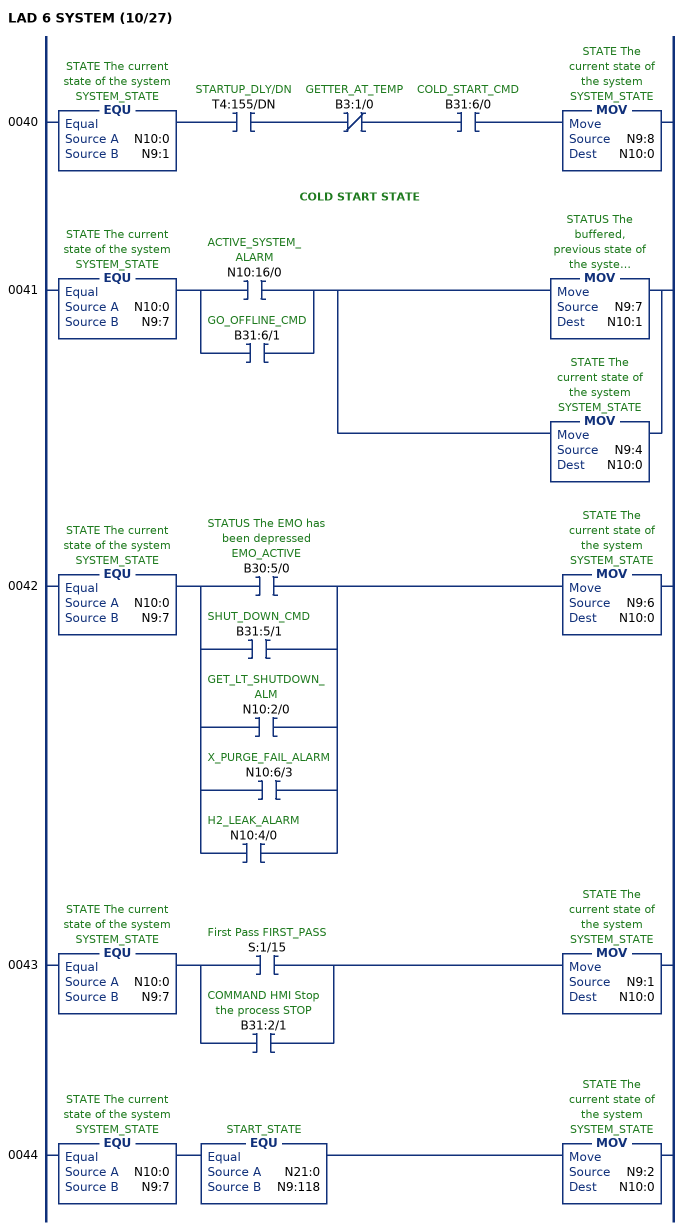
% Rung: 40 %
SOR EQU N10:0 N9:1 XIC T4:155/DN XIO B3:1/0 XIC B31:6/0 MOV N9:8 N10:0 EOR
%   N10:0  SYSTEM_STATE  "STATE The current state of the system" %
%   N9:1  SYSTEM_STANDBY  "STATE System Process" %
%   T4:155  STARTUP_DLY %
%   B3:1/0  GETTER_AT_TEMP %
%   B31:6/0  COLD_START_CMD %
%   N9:8  SYSTEM_SUPPLEMENTAL %
% Rung: 41 %
% TITLE: COLD START STATE %
SOR EQU N10:0 N9:7 BST XIC N10:16/0 NXB XIC B31:6/1 BND BST MOV N9:7 N10:1 NXB MOV N9:4 N10:0 BND EOR
%   N10:0  SYSTEM_STATE  "STATE The current state of the system" %
%   N9:7  SYSTEM_COLD_START %
%   N10:16/0  ACTIVE_SYSTEM_ALARM %
%   B31:6/1  GO_OFFLINE_CMD %
%   N10:1  SYSTEM_STATE_BUFFER  "STATUS The buffered, previous state of the system" %
%   N9:4  SYSTEM_ALARM  "STATE System Alarm" %
% Rung: 42 %
SOR EQU N10:0 N9:7 BST XIC B30:5/0 NXB XIC B31:5/1 NXB XIC N10:2/0 NXB XIC N10:6/3 NXB XIC N10:4/0 BND MOV N9:6 N10:0 EOR
%   N10:0  SYSTEM_STATE  "STATE The current state of the system" %
%   N9:7  SYSTEM_COLD_START %
%   B30:5/0  EMO_ACTIVE  "STATUS The EMO has been depressed" %
%   B31:5/1  SHUT_DOWN_CMD %
%   N10:2/0  GET_LT_SHUTDOWN_ALM %
%   N10:6/3  X_PURGE_FAIL_ALARM %
%   N10:4/0  H2_LEAK_ALARM %
%   N9:6  SYSTEM_PURGE %
% Rung: 43 %
SOR EQU N10:0 N9:7 BST XIC S:1/15 NXB XIC B31:2/1 BND MOV N9:1 N10:0 EOR
%   N10:0  SYSTEM_STATE  "STATE The current state of the system" %
%   N9:7  SYSTEM_COLD_START %
%   S:1/15  FIRST_PASS  "First Pass" %
%   B31:2/1  STOP  "COMMAND HMI Stop the process" %
%   N9:1  SYSTEM_STANDBY  "STATE System Process" %
% Rung: 44 %
SOR EQU N10:0 N9:7 EQU N21:0 N9:118 MOV N9:2 N10:0 EOR
%   N10:0  SYSTEM_STATE  "STATE The current state of the system" %
%   N9:7  SYSTEM_COLD_START %
%   N21:0  START_STATE %
%   N9:118  START_DONE %
%   N9:2  SYSTEM_PROCESS  "STATE System Process" %

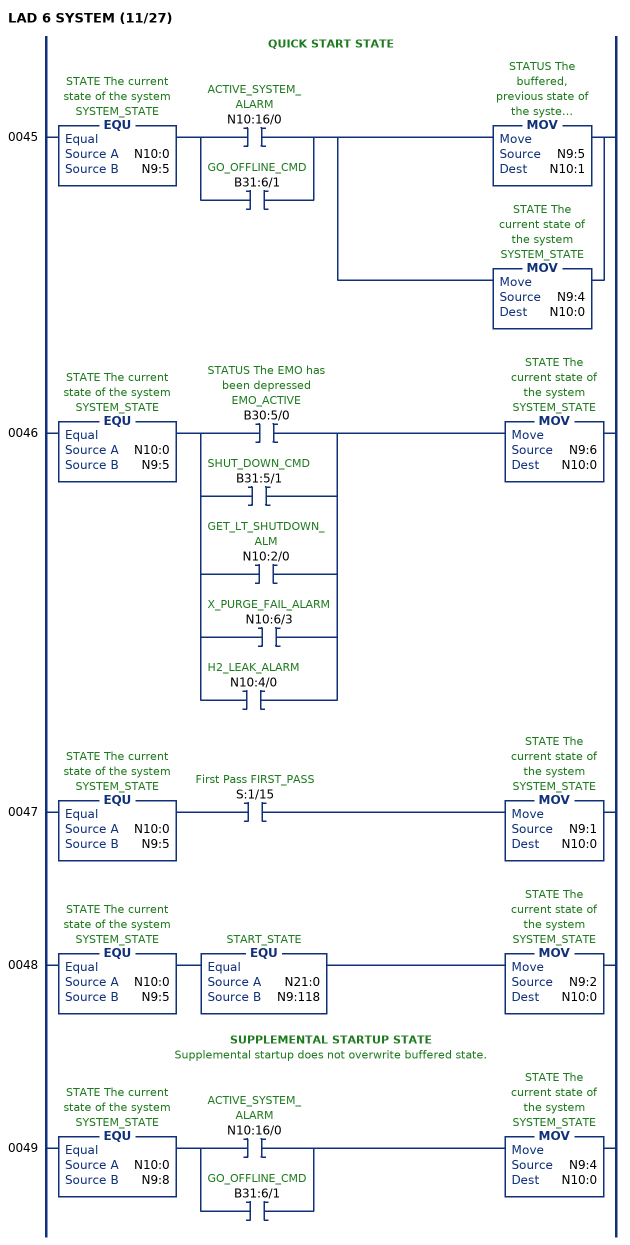
% Rung: 45 %
% TITLE: QUICK START STATE %
SOR EQU N10:0 N9:5 BST XIC N10:16/0 NXB XIC B31:6/1 BND BST MOV N9:5 N10:1 NXB MOV N9:4 N10:0 BND EOR
%   N10:0  SYSTEM_STATE  "STATE The current state of the system" %
%   N9:5  SYSTEM_QUICK_START %
%   N10:16/0  ACTIVE_SYSTEM_ALARM %
%   B31:6/1  GO_OFFLINE_CMD %
%   N10:1  SYSTEM_STATE_BUFFER  "STATUS The buffered, previous state of the system" %
%   N9:4  SYSTEM_ALARM  "STATE System Alarm" %
% Rung: 46 %
SOR EQU N10:0 N9:5 BST XIC B30:5/0 NXB XIC B31:5/1 NXB XIC N10:2/0 NXB XIC N10:6/3 NXB XIC N10:4/0 BND MOV N9:6 N10:0 EOR
%   N10:0  SYSTEM_STATE  "STATE The current state of the system" %
%   N9:5  SYSTEM_QUICK_START %
%   B30:5/0  EMO_ACTIVE  "STATUS The EMO has been depressed" %
%   B31:5/1  SHUT_DOWN_CMD %
%   N10:2/0  GET_LT_SHUTDOWN_ALM %
%   N10:6/3  X_PURGE_FAIL_ALARM %
%   N10:4/0  H2_LEAK_ALARM %
%   N9:6  SYSTEM_PURGE %
% Rung: 47 %
SOR EQU N10:0 N9:5 XIC S:1/15 MOV N9:1 N10:0 EOR
%   N10:0  SYSTEM_STATE  "STATE The current state of the system" %
%   N9:5  SYSTEM_QUICK_START %
%   S:1/15  FIRST_PASS  "First Pass" %
%   N9:1  SYSTEM_STANDBY  "STATE System Process" %
% Rung: 48 %
SOR EQU N10:0 N9:5 EQU N21:0 N9:118 MOV N9:2 N10:0 EOR
%   N10:0  SYSTEM_STATE  "STATE The current state of the system" %
%   N9:5  SYSTEM_QUICK_START %
%   N21:0  START_STATE %
%   N9:118  START_DONE %
%   N9:2  SYSTEM_PROCESS  "STATE System Process" %
% Rung: 49 %
% TITLE: SUPPLEMENTAL STARTUP STATE %
% Supplemental startup does not overwrite buffered state. %
SOR EQU N10:0 N9:8 BST XIC N10:16/0 NXB XIC B31:6/1 BND MOV N9:4 N10:0 EOR
%   N10:0  SYSTEM_STATE  "STATE The current state of the system" %
%   N9:8  SYSTEM_SUPPLEMENTAL %
%   N10:16/0  ACTIVE_SYSTEM_ALARM %
%   B31:6/1  GO_OFFLINE_CMD %
%   N9:4  SYSTEM_ALARM  "STATE System Alarm" %

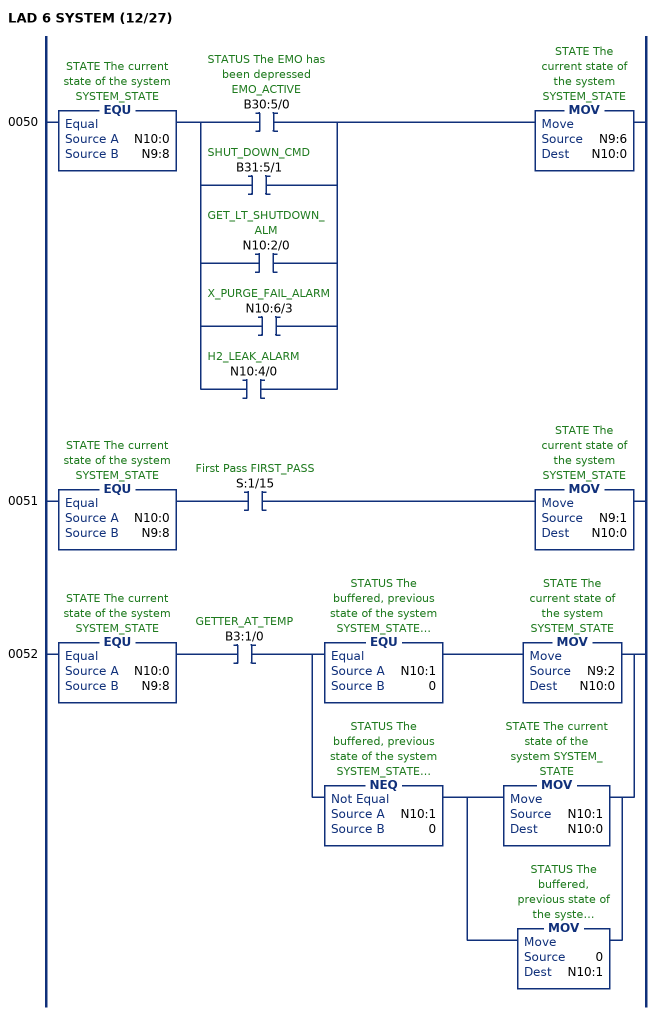
% Rung: 50 %
SOR EQU N10:0 N9:8 BST XIC B30:5/0 NXB XIC B31:5/1 NXB XIC N10:2/0 NXB XIC N10:6/3 NXB XIC N10:4/0 BND MOV N9:6 N10:0 EOR
%   N10:0  SYSTEM_STATE  "STATE The current state of the system" %
%   N9:8  SYSTEM_SUPPLEMENTAL %
%   B30:5/0  EMO_ACTIVE  "STATUS The EMO has been depressed" %
%   B31:5/1  SHUT_DOWN_CMD %
%   N10:2/0  GET_LT_SHUTDOWN_ALM %
%   N10:6/3  X_PURGE_FAIL_ALARM %
%   N10:4/0  H2_LEAK_ALARM %
%   N9:6  SYSTEM_PURGE %
% Rung: 51 %
SOR EQU N10:0 N9:8 XIC S:1/15 MOV N9:1 N10:0 EOR
%   N10:0  SYSTEM_STATE  "STATE The current state of the system" %
%   N9:8  SYSTEM_SUPPLEMENTAL %
%   S:1/15  FIRST_PASS  "First Pass" %
%   N9:1  SYSTEM_STANDBY  "STATE System Process" %
% Rung: 52 %
SOR EQU N10:0 N9:8 XIC B3:1/0 BST EQU N10:1 0 MOV N9:2 N10:0 NXB NEQ N10:1 0 BST MOV N10:1 N10:0 NXB MOV 0 N10:1 BND BND EOR
%   N10:0  SYSTEM_STATE  "STATE The current state of the system" %
%   N9:8  SYSTEM_SUPPLEMENTAL %
%   B3:1/0  GETTER_AT_TEMP %
%   N10:1  SYSTEM_STATE_BUFFER  "STATUS The buffered, previous state of the system" %
%   N9:2  SYSTEM_PROCESS  "STATE System Process" %

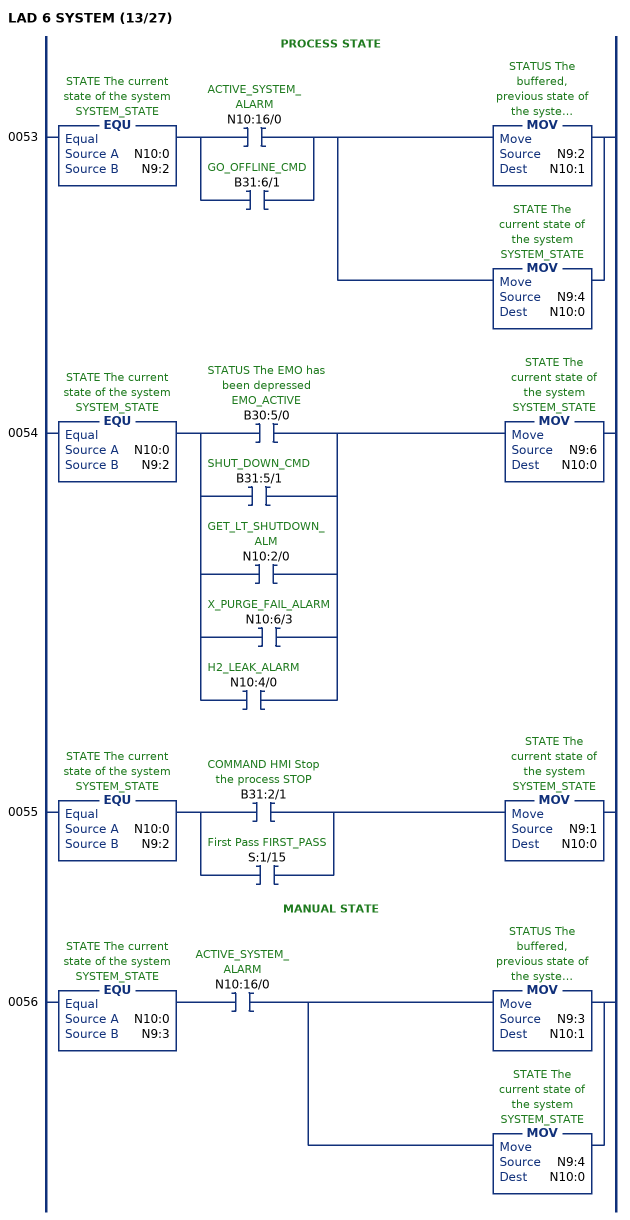
% Rung: 53 %
% TITLE: PROCESS STATE %
SOR EQU N10:0 N9:2 BST XIC N10:16/0 NXB XIC B31:6/1 BND BST MOV N9:2 N10:1 NXB MOV N9:4 N10:0 BND EOR
%   N10:0  SYSTEM_STATE  "STATE The current state of the system" %
%   N9:2  SYSTEM_PROCESS  "STATE System Process" %
%   N10:16/0  ACTIVE_SYSTEM_ALARM %
%   B31:6/1  GO_OFFLINE_CMD %
%   N10:1  SYSTEM_STATE_BUFFER  "STATUS The buffered, previous state of the system" %
%   N9:4  SYSTEM_ALARM  "STATE System Alarm" %
% Rung: 54 %
SOR EQU N10:0 N9:2 BST XIC B30:5/0 NXB XIC B31:5/1 NXB XIC N10:2/0 NXB XIC N10:6/3 NXB XIC N10:4/0 BND MOV N9:6 N10:0 EOR
%   N10:0  SYSTEM_STATE  "STATE The current state of the system" %
%   N9:2  SYSTEM_PROCESS  "STATE System Process" %
%   B30:5/0  EMO_ACTIVE  "STATUS The EMO has been depressed" %
%   B31:5/1  SHUT_DOWN_CMD %
%   N10:2/0  GET_LT_SHUTDOWN_ALM %
%   N10:6/3  X_PURGE_FAIL_ALARM %
%   N10:4/0  H2_LEAK_ALARM %
%   N9:6  SYSTEM_PURGE %
% Rung: 55 %
SOR EQU N10:0 N9:2 BST XIC B31:2/1 NXB XIC S:1/15 BND MOV N9:1 N10:0 EOR
%   N10:0  SYSTEM_STATE  "STATE The current state of the system" %
%   N9:2  SYSTEM_PROCESS  "STATE System Process" %
%   B31:2/1  STOP  "COMMAND HMI Stop the process" %
%   S:1/15  FIRST_PASS  "First Pass" %
%   N9:1  SYSTEM_STANDBY  "STATE System Process" %
% Rung: 56 %
% TITLE: MANUAL STATE %
SOR EQU N10:0 N9:3 XIC N10:16/0 BST MOV N9:3 N10:1 NXB MOV N9:4 N10:0 BND EOR
%   N10:0  SYSTEM_STATE  "STATE The current state of the system" %
%   N9:3  SYSTEM_MANUAL  "STATE System Manual" %
%   N10:16/0  ACTIVE_SYSTEM_ALARM %
%   N10:1  SYSTEM_STATE_BUFFER  "STATUS The buffered, previous state of the system" %
%   N9:4  SYSTEM_ALARM  "STATE System Alarm" %

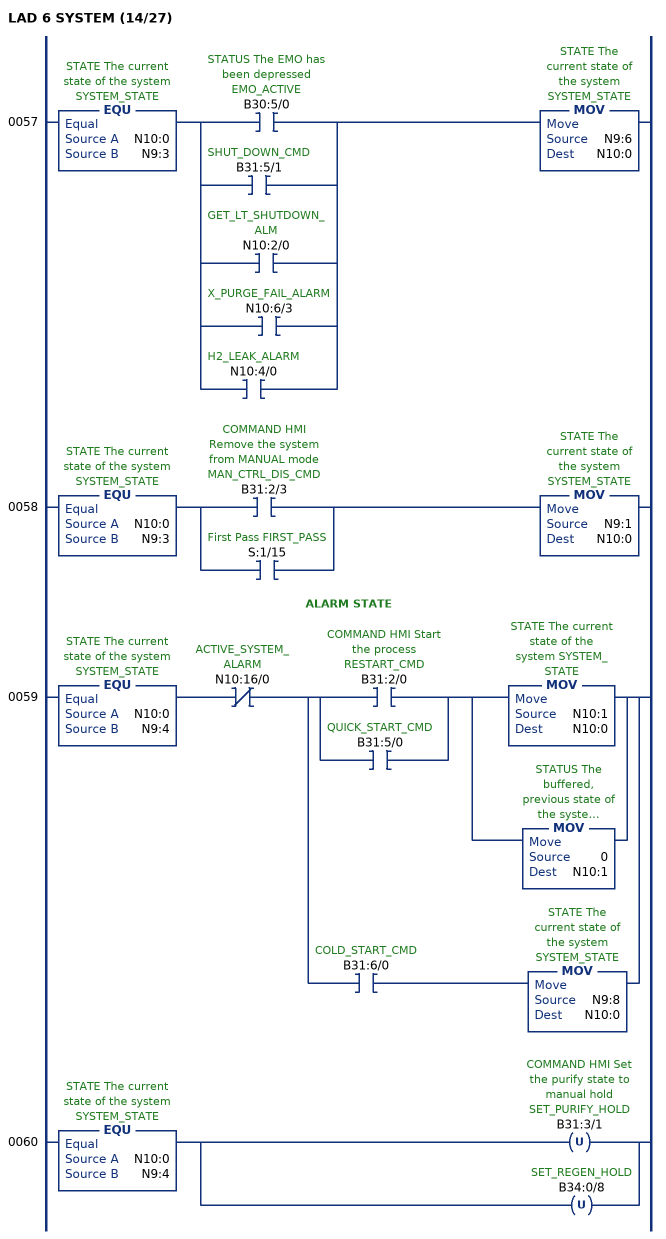
% Rung: 57 %
SOR EQU N10:0 N9:3 BST XIC B30:5/0 NXB XIC B31:5/1 NXB XIC N10:2/0 NXB XIC N10:6/3 NXB XIC N10:4/0 BND MOV N9:6 N10:0 EOR
%   N10:0  SYSTEM_STATE  "STATE The current state of the system" %
%   N9:3  SYSTEM_MANUAL  "STATE System Manual" %
%   B30:5/0  EMO_ACTIVE  "STATUS The EMO has been depressed" %
%   B31:5/1  SHUT_DOWN_CMD %
%   N10:2/0  GET_LT_SHUTDOWN_ALM %
%   N10:6/3  X_PURGE_FAIL_ALARM %
%   N10:4/0  H2_LEAK_ALARM %
%   N9:6  SYSTEM_PURGE %
% Rung: 58 %
SOR EQU N10:0 N9:3 BST XIC B31:2/3 NXB XIC S:1/15 BND MOV N9:1 N10:0 EOR
%   N10:0  SYSTEM_STATE  "STATE The current state of the system" %
%   N9:3  SYSTEM_MANUAL  "STATE System Manual" %
%   B31:2/3  MAN_CTRL_DIS_CMD  "COMMAND HMI Remove the system from MANUAL mode" %
%   S:1/15  FIRST_PASS  "First Pass" %
%   N9:1  SYSTEM_STANDBY  "STATE System Process" %
% Rung: 59 %
% TITLE: ALARM STATE %
SOR EQU N10:0 N9:4 XIO N10:16/0 BST BST XIC B31:2/0 NXB XIC B31:5/0 BND BST MOV N10:1 N10:0 NXB MOV 0 N10:1 BND NXB XIC B31:6/0 MOV N9:8 N10:0 BND EOR
%   N10:0  SYSTEM_STATE  "STATE The current state of the system" %
%   N9:4  SYSTEM_ALARM  "STATE System Alarm" %
%   N10:16/0  ACTIVE_SYSTEM_ALARM %
%   B31:2/0  RESTART_CMD  "COMMAND HMI Start the process" %
%   B31:5/0  QUICK_START_CMD %
%   N10:1  SYSTEM_STATE_BUFFER  "STATUS The buffered, previous state of the system" %
%   B31:6/0  COLD_START_CMD %
%   N9:8  SYSTEM_SUPPLEMENTAL %
% Rung: 60 %
SOR EQU N10:0 N9:4 BST OTU B31:3/1 NXB OTU B34:0/8 BND EOR
%   N10:0  SYSTEM_STATE  "STATE The current state of the system" %
%   N9:4  SYSTEM_ALARM  "STATE System Alarm" %
%   B31:3/1  SET_PURIFY_HOLD  "COMMAND HMI Set the purify state to manual hold" %
%   B34:0/8  SET_REGEN_HOLD %

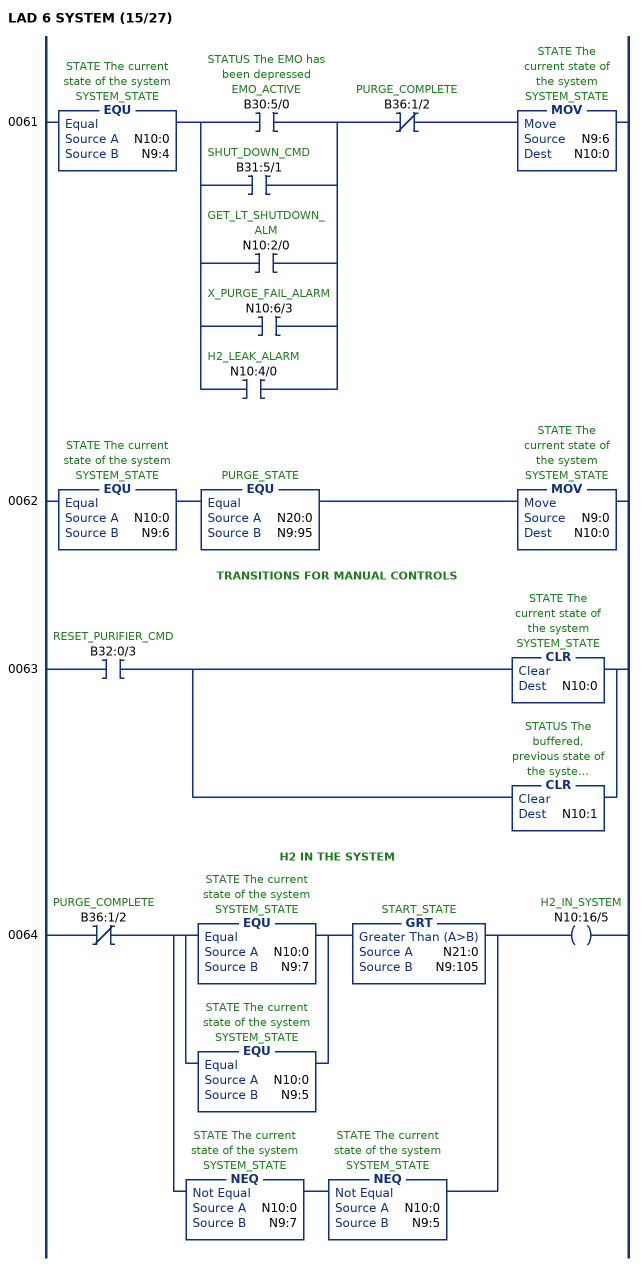
% Rung: 61 %
SOR EQU N10:0 N9:4 BST XIC B30:5/0 NXB XIC B31:5/1 NXB XIC N10:2/0 NXB XIC N10:6/3 NXB XIC N10:4/0 BND XIO B36:1/2 MOV N9:6 N10:0 EOR
%   N10:0  SYSTEM_STATE  "STATE The current state of the system" %
%   N9:4  SYSTEM_ALARM  "STATE System Alarm" %
%   B30:5/0  EMO_ACTIVE  "STATUS The EMO has been depressed" %
%   B31:5/1  SHUT_DOWN_CMD %
%   N10:2/0  GET_LT_SHUTDOWN_ALM %
%   N10:6/3  X_PURGE_FAIL_ALARM %
%   N10:4/0  H2_LEAK_ALARM %
%   B36:1/2  PURGE_COMPLETE %
%   N9:6  SYSTEM_PURGE %
% Rung: 62 %
SOR EQU N10:0 N9:6 EQU N20:0 N9:95 MOV N9:0 N10:0 EOR
%   N10:0  SYSTEM_STATE  "STATE The current state of the system" %
%   N9:6  SYSTEM_PURGE %
%   N20:0  PURGE_STATE %
%   N9:95  PURGE_DONE %
%   N9:0  SYSTEM_OFFLINE %
% Rung: 63 %
% TITLE: TRANSITIONS FOR MANUAL CONTROLS %
SOR XIC B32:0/3 BST CLR N10:0 NXB CLR N10:1 BND EOR
%   B32:0/3  RESET_PURIFIER_CMD %
%   N10:0  SYSTEM_STATE  "STATE The current state of the system" %
%   N10:1  SYSTEM_STATE_BUFFER  "STATUS The buffered, previous state of the system" %
% Rung: 64 %
% TITLE: H2 IN THE SYSTEM %
SOR XIO B36:1/2 BST BST EQU N10:0 N9:7 NXB EQU N10:0 N9:5 BND GRT N21:0 N9:105 NXB NEQ N10:0 N9:7 NEQ N10:0 N9:5 BND OTE N10:16/5 EOR
%   B36:1/2  PURGE_COMPLETE %
%   N10:0  SYSTEM_STATE  "STATE The current state of the system" %
%   N9:7  SYSTEM_COLD_START %
%   N9:5  SYSTEM_QUICK_START %
%   N21:0  START_STATE %
%   N9:105  START_VENT_ALL %
%   N10:16/5  H2_IN_SYSTEM %

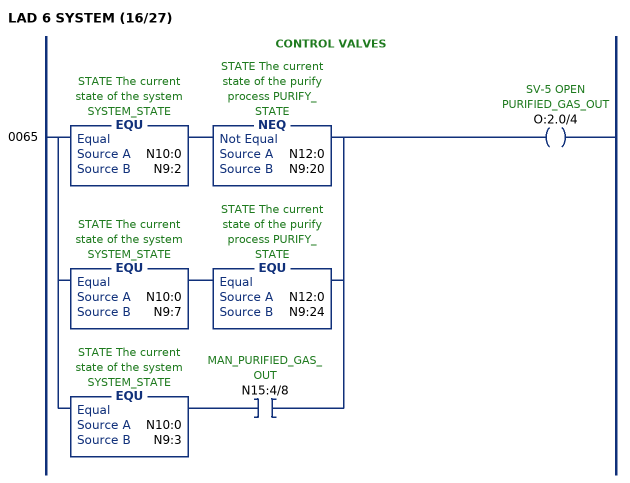
% Rung: 65 %
% TITLE: CONTROL VALVES %
SOR BST EQU N10:0 N9:2 NEQ N12:0 N9:20 NXB EQU N10:0 N9:7 EQU N12:0 N9:24 NXB EQU N10:0 N9:3 XIC N15:4/8 BND OTE O:2.0/4 EOR
%   N10:0  SYSTEM_STATE  "STATE The current state of the system" %
%   N9:2  SYSTEM_PROCESS  "STATE System Process" %
%   N12:0  PURIFY_STATE  "STATE The current state of the purify process" %
%   N9:20  PURIFY_STANDBY  "STATE Purify Standby" %
%   N9:7  SYSTEM_COLD_START %
%   N9:24  PURIFY_OVERLAP  "STATE Puriify Overlap" %
%   N9:3  SYSTEM_MANUAL  "STATE System Manual" %
%   N15:4/8  MAN_PURIFIED_GAS_OUT %
%   O:2.0/4  PURIFIED_GAS_OUT  "SV-5 OPEN" %

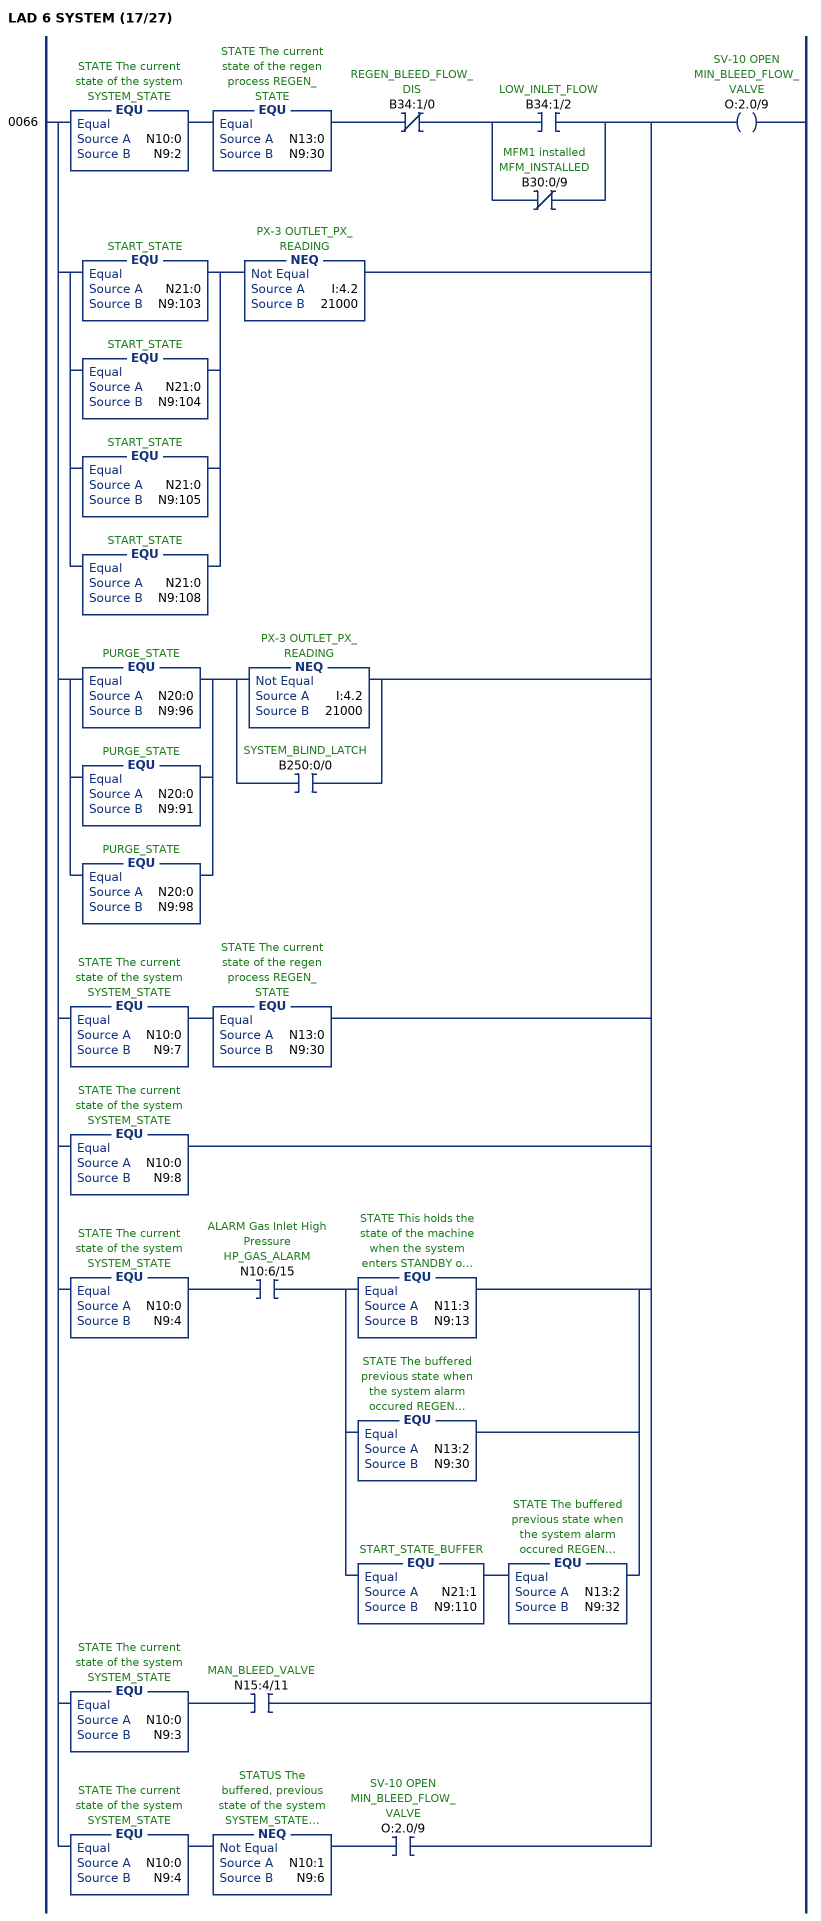
% Rung: 66 %
SOR BST EQU N10:0 N9:2 EQU N13:0 N9:30 XIO B34:1/0 BST XIC B34:1/2 NXB XIO B30:0/9 BND NXB BST EQU N21:0 N9:103 NXB EQU N21:0 N9:104 NXB EQU N21:0 N9:105 NXB EQU N21:0 N9:108 BND NEQ I:4.2 21000 NXB BST EQU N20:0 N9:96 NXB EQU N20:0 N9:91 NXB EQU N20:0 N9:98 BND BST NEQ I:4.2 21000 NXB XIC B250:0/0 BND NXB EQU N10:0 N9:7 EQU N13:0 N9:30 NXB EQU N10:0 N9:8 NXB EQU N10:0 N9:4 XIC N10:6/15 BST EQU N11:3 N9:13 NXB EQU N13:2 N9:30 NXB EQU N21:1 N9:110 EQU N13:2 N9:32 BND NXB EQU N10:0 N9:3 XIC N15:4/11 NXB EQU N10:0 N9:4 NEQ N10:1 N9:6 XIC O:2.0/9 BND OTE O:2.0/9 EOR
%   N10:0  SYSTEM_STATE  "STATE The current state of the system" %
%   N9:2  SYSTEM_PROCESS  "STATE System Process" %
%   N13:0  REGEN_STATE  "STATE The current state of the regen process" %
%   N9:30  REGEN_STANDBY  "STATE Regen Standby" %
%   B34:1/0  REGEN_BLEED_FLOW_DIS %
%   B34:1/2  LOW_INLET_FLOW %
%   B30:0/9  MFM_INSTALLED  "MFM1 installed" %
%   N21:0  START_STATE %
%   N9:103  START_VENT_GET_1 %
%   N9:104  START_HEAT_GETTER %
%   N9:105  START_VENT_ALL %
%   N9:108  START_VENT_GET_2 %
%   I:4.2  OUTLET_PX_READING  "PX-3" %
%   N20:0  PURGE_STATE %
%   N9:96  PURGE_VENT_GETTER %
%   N9:91  PURGE_INIT_VENT %
%   N9:98  PURGE_VENT_GET_2 %
%   B250:0/0  SYSTEM_BLIND_LATCH %
%   N9:7  SYSTEM_COLD_START %
%   N9:8  SYSTEM_SUPPLEMENTAL %
%   N9:4  SYSTEM_ALARM  "STATE System Alarm" %
%   N10:6/15  HP_GAS_ALARM  "ALARM Gas Inlet High Pressure" %
%   N11:3  PROC_STATE_BUFFER  "STATE This holds the state of the machine when the system enters STANDBY or ALARM" %
%   N9:13  PROC_OVERLAP  "STATE Process Purify Overlap" %
%   N13:2  REGEN_SYSTEM_BUFFER  "STATE The buffered previous state when the system alarm occured" %
%   N21:1  START_STATE_BUFFER %
%   N9:110  START_REG_VENT %
%   N9:32  REGEN_VENT  "STATE Regen Vent" %
%   N9:3  SYSTEM_MANUAL  "STATE System Manual" %
%   N15:4/11  MAN_BLEED_VALVE %
%   N10:1  SYSTEM_STATE_BUFFER  "STATUS The buffered, previous state of the system" %
%   N9:6  SYSTEM_PURGE %
%   O:2.0/9  MIN_BLEED_FLOW_VALVE  "SV-10 OPEN" %

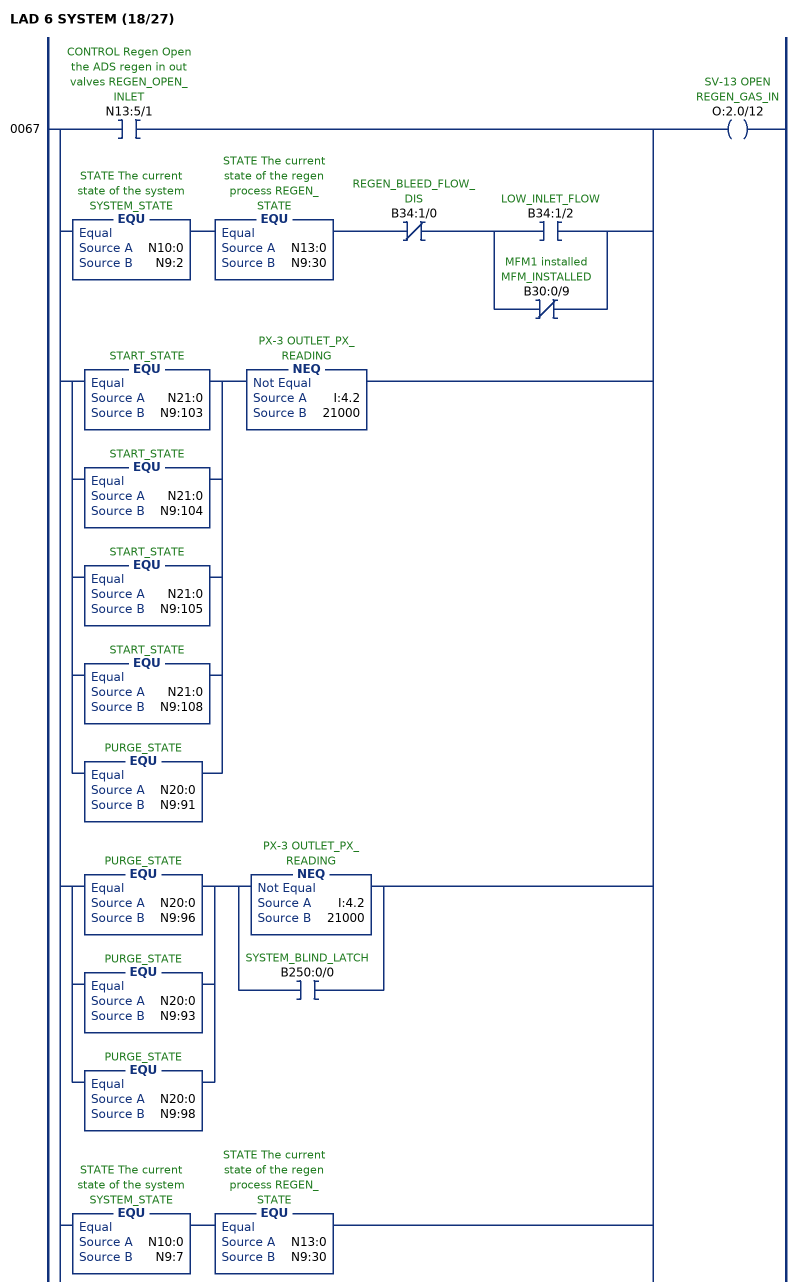

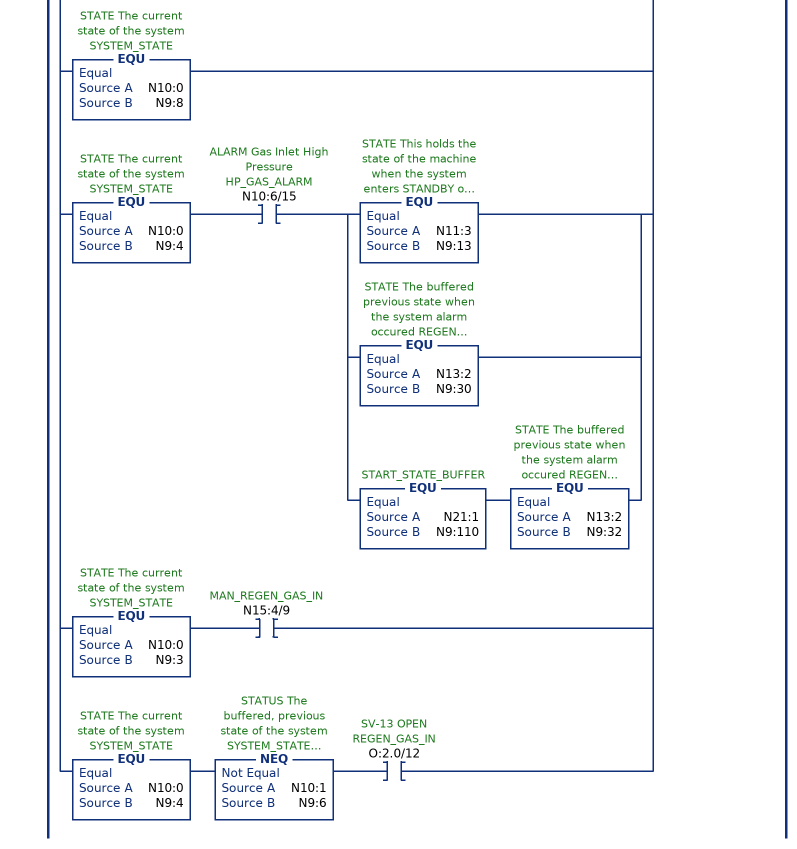
% Rung: 67 %
SOR BST XIC N13:5/1 NXB EQU N10:0 N9:2 EQU N13:0 N9:30 XIO B34:1/0 BST XIC B34:1/2 NXB XIO B30:0/9 BND NXB BST EQU N21:0 N9:103 NXB EQU N21:0 N9:104 NXB EQU N21:0 N9:105 NXB EQU N21:0 N9:108 NXB EQU N20:0 N9:91 BND NEQ I:4.2 21000 NXB BST EQU N20:0 N9:96 NXB EQU N20:0 N9:93 NXB EQU N20:0 N9:98 BND BST NEQ I:4.2 21000 NXB XIC B250:0/0 BND NXB EQU N10:0 N9:7 EQU N13:0 N9:30 NXB EQU N10:0 N9:8 NXB EQU N10:0 N9:4 XIC N10:6/15 BST EQU N11:3 N9:13 NXB EQU N13:2 N9:30 NXB EQU N21:1 N9:110 EQU N13:2 N9:32 BND NXB EQU N10:0 N9:3 XIC N15:4/9 NXB EQU N10:0 N9:4 NEQ N10:1 N9:6 XIC O:2.0/12 BND OTE O:2.0/12 EOR
%   N13:5/1  REGEN_OPEN_INLET  "CONTROL Regen Open the ADS regen in out valves" %
%   N10:0  SYSTEM_STATE  "STATE The current state of the system" %
%   N9:2  SYSTEM_PROCESS  "STATE System Process" %
%   N13:0  REGEN_STATE  "STATE The current state of the regen process" %
%   N9:30  REGEN_STANDBY  "STATE Regen Standby" %
%   B34:1/0  REGEN_BLEED_FLOW_DIS %
%   B34:1/2  LOW_INLET_FLOW %
%   B30:0/9  MFM_INSTALLED  "MFM1 installed" %
%   N21:0  START_STATE %
%   N9:103  START_VENT_GET_1 %
%   N9:104  START_HEAT_GETTER %
%   N9:105  START_VENT_ALL %
%   N9:108  START_VENT_GET_2 %
%   N20:0  PURGE_STATE %
%   N9:91  PURGE_INIT_VENT %
%   I:4.2  OUTLET_PX_READING  "PX-3" %
%   N9:96  PURGE_VENT_GETTER %
%   N9:93  PURGE_BACKFILL %
%   N9:98  PURGE_VENT_GET_2 %
%   B250:0/0  SYSTEM_BLIND_LATCH %
%   N9:7  SYSTEM_COLD_START %
%   N9:8  SYSTEM_SUPPLEMENTAL %
%   N9:4  SYSTEM_ALARM  "STATE System Alarm" %
%   N10:6/15  HP_GAS_ALARM  "ALARM Gas Inlet High Pressure" %
%   N11:3  PROC_STATE_BUFFER  "STATE This holds the state of the machine when the system enters STANDBY or ALARM" %
%   N9:13  PROC_OVERLAP  "STATE Process Purify Overlap" %
%   N13:2  REGEN_SYSTEM_BUFFER  "STATE The buffered previous state when the system alarm occured" %
%   N21:1  START_STATE_BUFFER %
%   N9:110  START_REG_VENT %
%   N9:32  REGEN_VENT  "STATE Regen Vent" %
%   N9:3  SYSTEM_MANUAL  "STATE System Manual" %
%   N15:4/9  MAN_REGEN_GAS_IN %
%   N10:1  SYSTEM_STATE_BUFFER  "STATUS The buffered, previous state of the system" %
%   N9:6  SYSTEM_PURGE %
%   O:2.0/12  REGEN_GAS_IN  "SV-13 OPEN" %

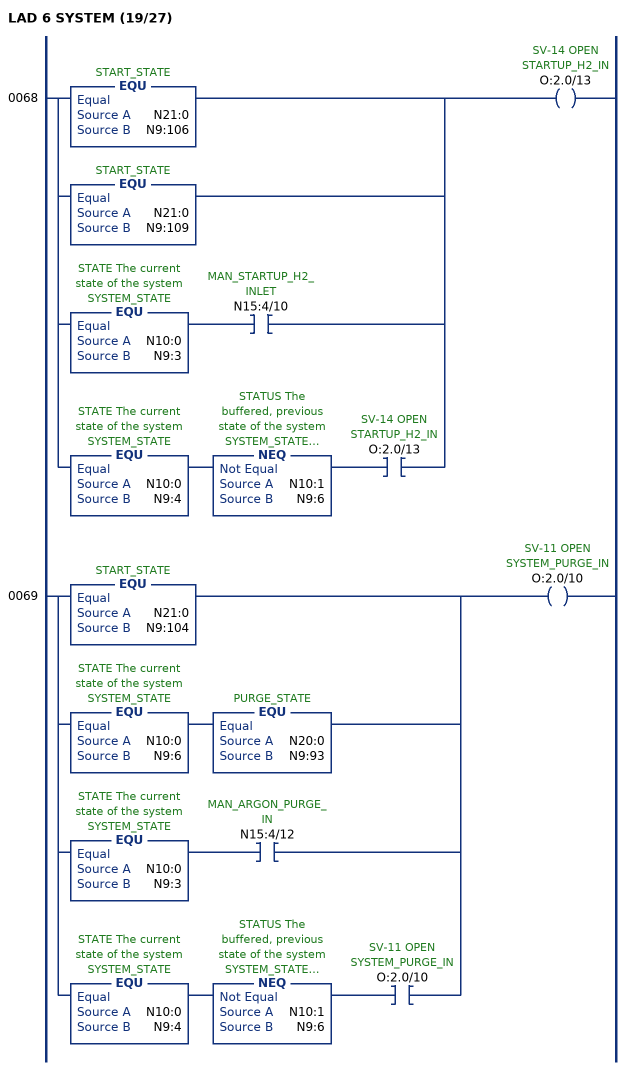
% Rung: 68 %
SOR BST BST EQU N21:0 N9:106 NXB EQU N21:0 N9:109 BND NXB EQU N10:0 N9:3 XIC N15:4/10 NXB EQU N10:0 N9:4 NEQ N10:1 N9:6 XIC O:2.0/13 BND OTE O:2.0/13 EOR
%   N21:0  START_STATE %
%   N9:106  START_BACKFILL_1 %
%   N9:109  START_BKFL_2 %
%   N10:0  SYSTEM_STATE  "STATE The current state of the system" %
%   N9:3  SYSTEM_MANUAL  "STATE System Manual" %
%   N15:4/10  MAN_STARTUP_H2_INLET %
%   N9:4  SYSTEM_ALARM  "STATE System Alarm" %
%   N10:1  SYSTEM_STATE_BUFFER  "STATUS The buffered, previous state of the system" %
%   N9:6  SYSTEM_PURGE %
%   O:2.0/13  STARTUP_H2_IN  "SV-14 OPEN" %
% Rung: 69 %
SOR BST EQU N21:0 N9:104 NXB EQU N10:0 N9:6 EQU N20:0 N9:93 NXB EQU N10:0 N9:3 XIC N15:4/12 NXB EQU N10:0 N9:4 NEQ N10:1 N9:6 XIC O:2.0/10 BND OTE O:2.0/10 EOR
%   N21:0  START_STATE %
%   N9:104  START_HEAT_GETTER %
%   N10:0  SYSTEM_STATE  "STATE The current state of the system" %
%   N9:6  SYSTEM_PURGE %
%   N20:0  PURGE_STATE %
%   N9:93  PURGE_BACKFILL %
%   N9:3  SYSTEM_MANUAL  "STATE System Manual" %
%   N15:4/12  MAN_ARGON_PURGE_IN %
%   N9:4  SYSTEM_ALARM  "STATE System Alarm" %
%   N10:1  SYSTEM_STATE_BUFFER  "STATUS The buffered, previous state of the system" %
%   O:2.0/10  SYSTEM_PURGE_IN  "SV-11 OPEN" %

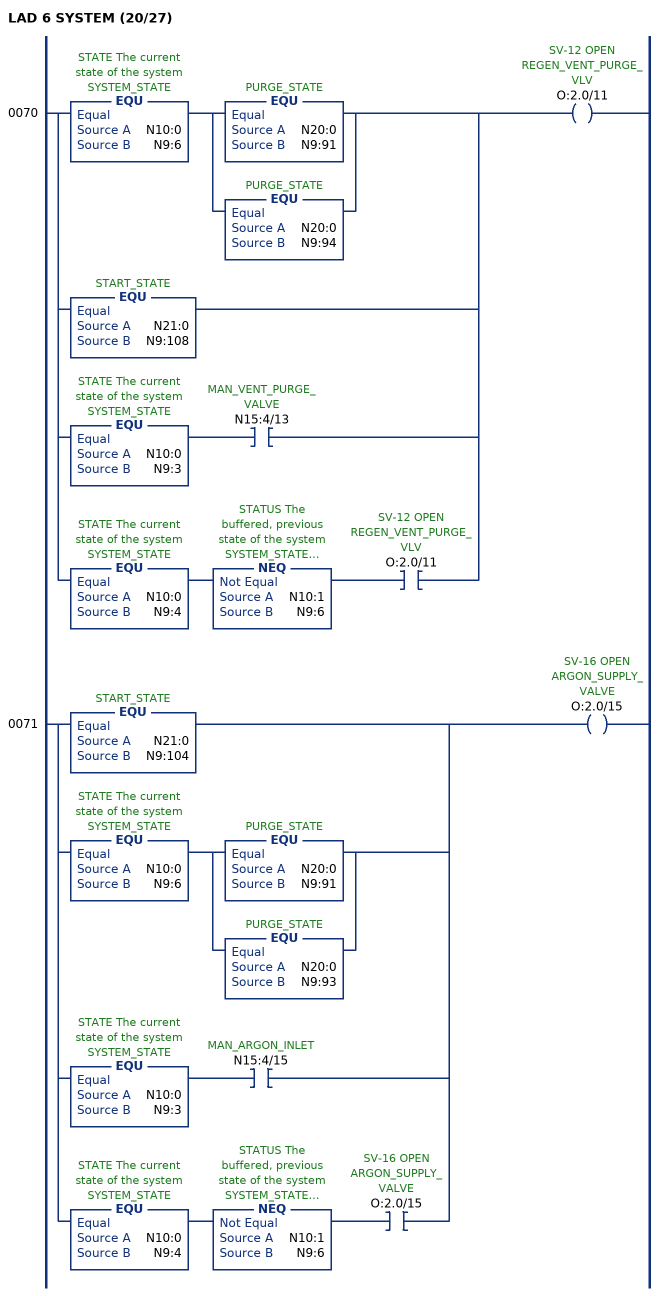
% Rung: 70 %
SOR BST EQU N10:0 N9:6 BST EQU N20:0 N9:91 NXB EQU N20:0 N9:94 BND NXB EQU N21:0 N9:108 NXB EQU N10:0 N9:3 XIC N15:4/13 NXB EQU N10:0 N9:4 NEQ N10:1 N9:6 XIC O:2.0/11 BND OTE O:2.0/11 EOR
%   N10:0  SYSTEM_STATE  "STATE The current state of the system" %
%   N9:6  SYSTEM_PURGE %
%   N20:0  PURGE_STATE %
%   N9:91  PURGE_INIT_VENT %
%   N9:94  PURGE_FINAL_VENT %
%   N21:0  START_STATE %
%   N9:108  START_VENT_GET_2 %
%   N9:3  SYSTEM_MANUAL  "STATE System Manual" %
%   N15:4/13  MAN_VENT_PURGE_VALVE %
%   N9:4  SYSTEM_ALARM  "STATE System Alarm" %
%   N10:1  SYSTEM_STATE_BUFFER  "STATUS The buffered, previous state of the system" %
%   O:2.0/11  REGEN_VENT_PURGE_VLV  "SV-12 OPEN" %
% Rung: 71 %
SOR BST EQU N21:0 N9:104 NXB EQU N10:0 N9:6 BST EQU N20:0 N9:91 NXB EQU N20:0 N9:93 BND NXB EQU N10:0 N9:3 XIC N15:4/15 NXB EQU N10:0 N9:4 NEQ N10:1 N9:6 XIC O:2.0/15 BND OTE O:2.0/15 EOR
%   N21:0  START_STATE %
%   N9:104  START_HEAT_GETTER %
%   N10:0  SYSTEM_STATE  "STATE The current state of the system" %
%   N9:6  SYSTEM_PURGE %
%   N20:0  PURGE_STATE %
%   N9:91  PURGE_INIT_VENT %
%   N9:93  PURGE_BACKFILL %
%   N9:3  SYSTEM_MANUAL  "STATE System Manual" %
%   N15:4/15  MAN_ARGON_INLET %
%   N9:4  SYSTEM_ALARM  "STATE System Alarm" %
%   N10:1  SYSTEM_STATE_BUFFER  "STATUS The buffered, previous state of the system" %
%   O:2.0/15  ARGON_SUPPLY_VALVE  "SV-16 OPEN" %

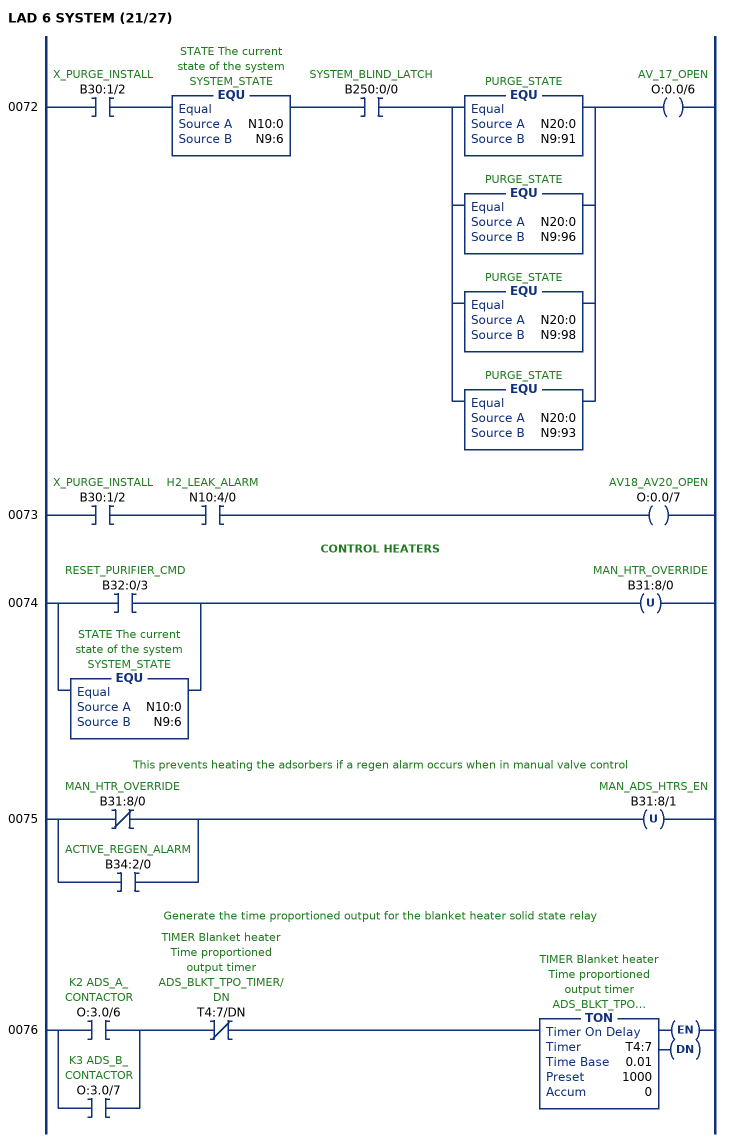
% Rung: 72 %
SOR XIC B30:1/2 EQU N10:0 N9:6 XIC B250:0/0 BST EQU N20:0 N9:91 NXB EQU N20:0 N9:96 NXB EQU N20:0 N9:98 NXB EQU N20:0 N9:93 BND OTE O:0.0/6 EOR
%   B30:1/2  X_PURGE_INSTALL %
%   N10:0  SYSTEM_STATE  "STATE The current state of the system" %
%   N9:6  SYSTEM_PURGE %
%   B250:0/0  SYSTEM_BLIND_LATCH %
%   N20:0  PURGE_STATE %
%   N9:91  PURGE_INIT_VENT %
%   N9:96  PURGE_VENT_GETTER %
%   N9:98  PURGE_VENT_GET_2 %
%   N9:93  PURGE_BACKFILL %
%   O:0.0/6  AV_17_OPEN %
% Rung: 73 %
SOR XIC B30:1/2 XIC N10:4/0 OTE O:0.0/7 EOR
%   B30:1/2  X_PURGE_INSTALL %
%   N10:4/0  H2_LEAK_ALARM %
%   O:0.0/7  AV18_AV20_OPEN %
% Rung: 74 %
% TITLE: CONTROL HEATERS %
SOR BST XIC B32:0/3 NXB EQU N10:0 N9:6 BND OTU B31:8/0 EOR
%   B32:0/3  RESET_PURIFIER_CMD %
%   N10:0  SYSTEM_STATE  "STATE The current state of the system" %
%   N9:6  SYSTEM_PURGE %
%   B31:8/0  MAN_HTR_OVERRIDE %
% Rung: 75 %
% This prevents heating the adsorbers if a regen alarm occurs when in manual valve control %
SOR BST XIO B31:8/0 NXB XIC B34:2/0 BND OTU B31:8/1 EOR
%   B31:8/0  MAN_HTR_OVERRIDE %
%   B34:2/0  ACTIVE_REGEN_ALARM %
%   B31:8/1  MAN_ADS_HTRS_EN %
% Rung: 76 %
% Generate the time proportioned output for the blanket heater solid state relay %
SOR BST XIC O:3.0/6 NXB XIC O:3.0/7 BND XIO T4:7/DN TON T4:7 0.01 1000 0 EOR
%   O:3.0/6  ADS_A_CONTACTOR  "K2" %
%   O:3.0/7  ADS_B_CONTACTOR  "K3" %
%   T4:7  ADS_BLKT_TPO_TIMER  "TIMER Blanket heater Time proportioned output timer" %

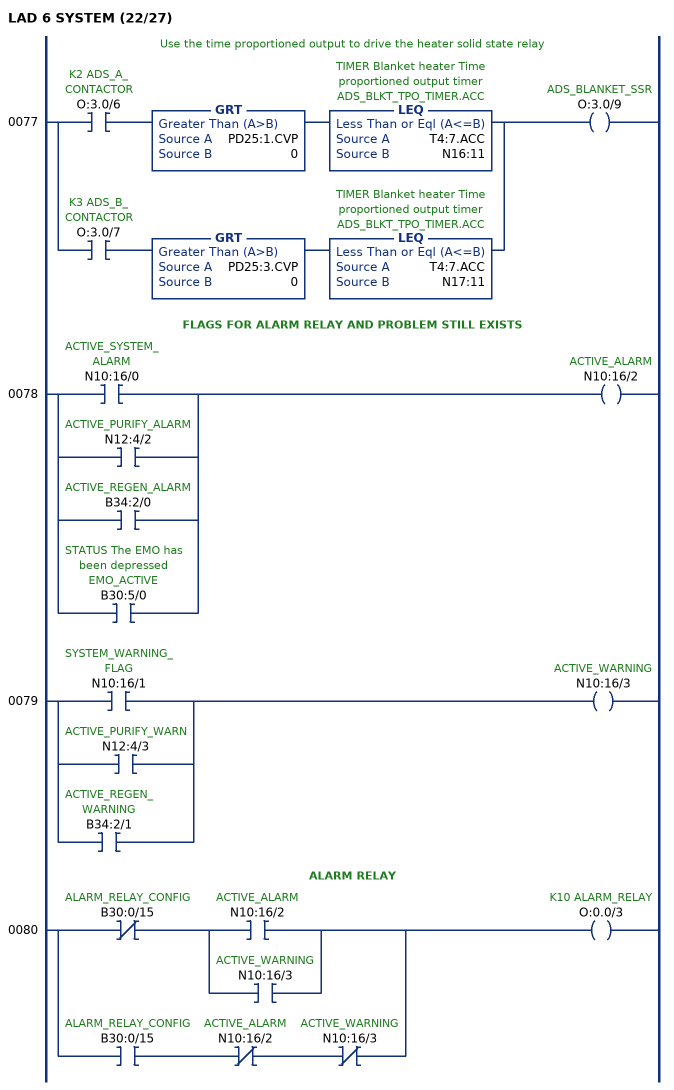
% Rung: 77 %
% Use the time proportioned output to drive the heater solid state relay %
SOR BST XIC O:3.0/6 GRT PD25:1.CVP 0 LEQ T4:7.ACC N16:11 NXB XIC O:3.0/7 GRT PD25:3.CVP 0 LEQ T4:7.ACC N17:11 BND OTE O:3.0/9 EOR
%   O:3.0/6  ADS_A_CONTACTOR  "K2" %
%   T4:7  ADS_BLKT_TPO_TIMER  "TIMER Blanket heater Time proportioned output timer" %
%   N16:11  ADS_A_BLNKT_OUTPUT  "CONTROL ADS A Blanket output (percent)" %
%   O:3.0/7  ADS_B_CONTACTOR  "K3" %
%   N17:11  ADS_B_BLNKT_OUTPUT  "CONTROL ADS A Blanket output" %
%   O:3.0/9  ADS_BLANKET_SSR %
% Rung: 78 %
% TITLE: FLAGS FOR ALARM RELAY AND PROBLEM STILL EXISTS %
SOR BST XIC N10:16/0 NXB XIC N12:4/2 NXB XIC B34:2/0 NXB XIC B30:5/0 BND OTE N10:16/2 EOR
%   N10:16/0  ACTIVE_SYSTEM_ALARM %
%   N12:4/2  ACTIVE_PURIFY_ALARM %
%   B34:2/0  ACTIVE_REGEN_ALARM %
%   B30:5/0  EMO_ACTIVE  "STATUS The EMO has been depressed" %
%   N10:16/2  ACTIVE_ALARM %
% Rung: 79 %
SOR BST XIC N10:16/1 NXB XIC N12:4/3 NXB XIC B34:2/1 BND OTE N10:16/3 EOR
%   N10:16/1  SYSTEM_WARNING_FLAG %
%   N12:4/3  ACTIVE_PURIFY_WARN %
%   B34:2/1  ACTIVE_REGEN_WARNING %
%   N10:16/3  ACTIVE_WARNING %
% Rung: 80 %
% TITLE: ALARM RELAY %
SOR BST XIO B30:0/15 BST XIC N10:16/2 NXB XIC N10:16/3 BND NXB XIC B30:0/15 XIO N10:16/2 XIO N10:16/3 BND OTE O:0.0/3 EOR
%   B30:0/15  ALARM_RELAY_CONFIG %
%   N10:16/2  ACTIVE_ALARM %
%   N10:16/3  ACTIVE_WARNING %
%   O:0.0/3  ALARM_RELAY  "K10" %

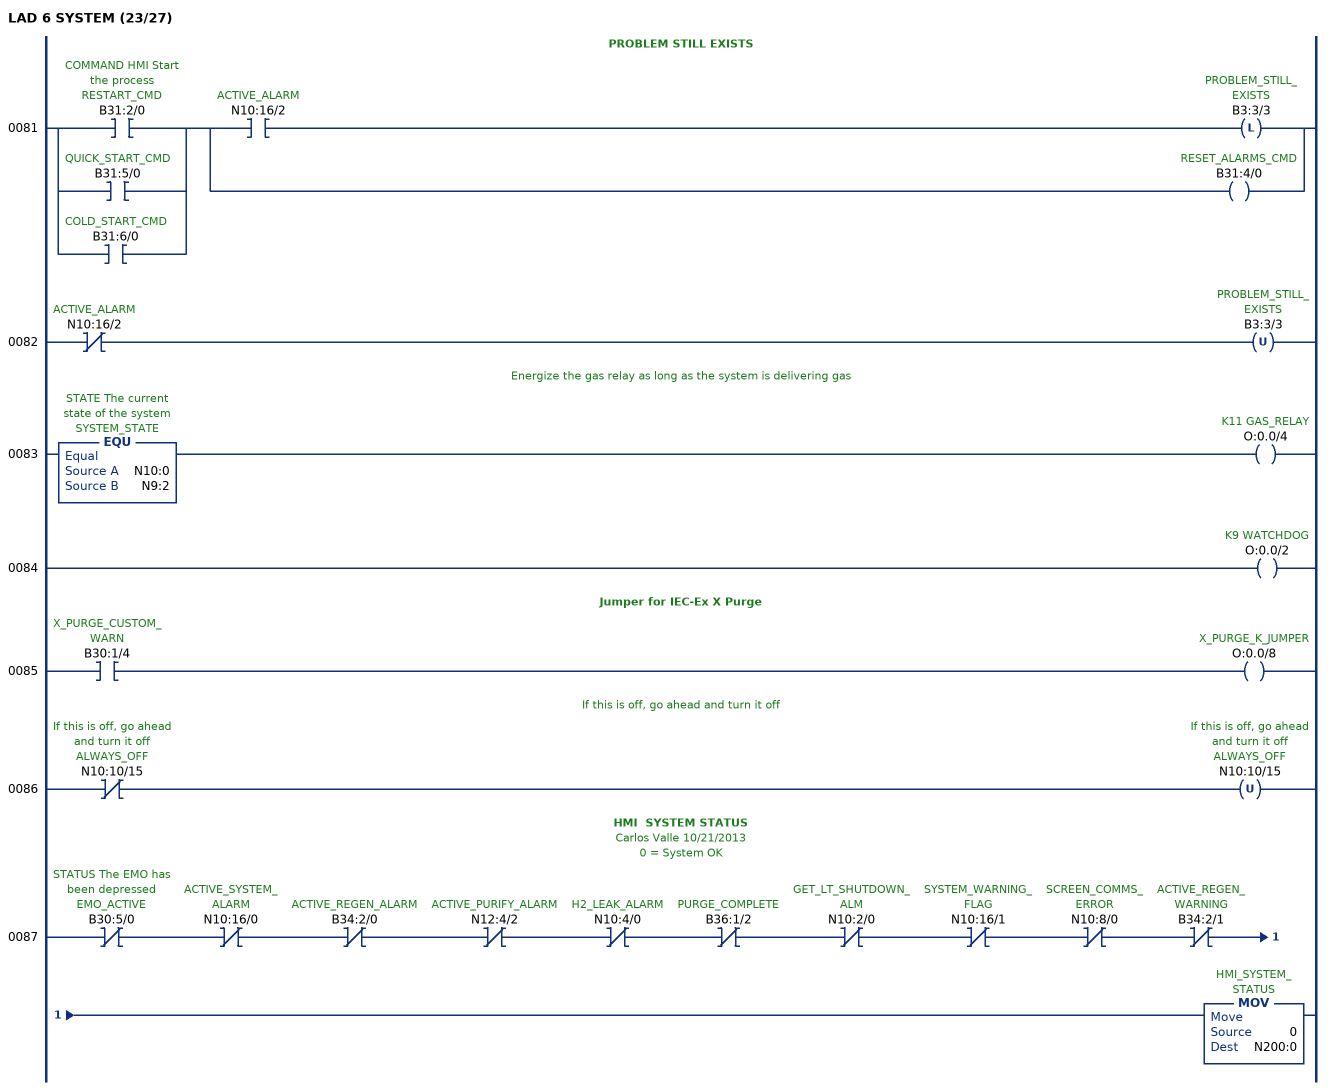
% Rung: 81 %
% TITLE: PROBLEM STILL EXISTS %
SOR BST XIC B31:2/0 NXB XIC B31:5/0 NXB XIC B31:6/0 BND BST XIC N10:16/2 OTL B3:3/3 NXB OTE B31:4/0 BND EOR
%   B31:2/0  RESTART_CMD  "COMMAND HMI Start the process" %
%   B31:5/0  QUICK_START_CMD %
%   B31:6/0  COLD_START_CMD %
%   N10:16/2  ACTIVE_ALARM %
%   B3:3/3  PROBLEM_STILL_EXISTS %
%   B31:4/0  RESET_ALARMS_CMD %
% Rung: 82 %
SOR XIO N10:16/2 OTU B3:3/3 EOR
%   N10:16/2  ACTIVE_ALARM %
%   B3:3/3  PROBLEM_STILL_EXISTS %
% Rung: 83 %
% Energize the gas relay as long as the system is delivering gas %
SOR EQU N10:0 N9:2 OTE O:0.0/4 EOR
%   N10:0  SYSTEM_STATE  "STATE The current state of the system" %
%   N9:2  SYSTEM_PROCESS  "STATE System Process" %
%   O:0.0/4  GAS_RELAY  "K11" %
% Rung: 84 %
SOR OTE O:0.0/2 EOR
%   O:0.0/2  WATCHDOG  "K9" %
% Rung: 85 %
% TITLE: Jumper for IEC-Ex X Purge %
SOR XIC B30:1/4 OTE O:0.0/8 EOR
%   B30:1/4  X_PURGE_CUSTOM_WARN %
%   O:0.0/8  X_PURGE_K_JUMPER %
% Rung: 86 %
% If this is off, go ahead and turn it off %
SOR XIO N10:10/15 OTU N10:10/15 EOR
%   N10:10/15  ALWAYS_OFF  "If this is off, go ahead and turn it off" %
% Rung: 87 %
% TITLE: HMI  SYSTEM STATUS %
% Carlos Valle 10/21/2013
% 0 = System OK %
SOR XIO B30:5/0 XIO N10:16/0 XIO B34:2/0 XIO N12:4/2 XIO N10:4/0 XIO B36:1/2 XIO N10:2/0 XIO N10:16/1 XIO N10:8/0 XIO B34:2/1 MOV 0 N200:0 EOR
%   B30:5/0  EMO_ACTIVE  "STATUS The EMO has been depressed" %
%   N10:16/0  ACTIVE_SYSTEM_ALARM %
%   B34:2/0  ACTIVE_REGEN_ALARM %
%   N12:4/2  ACTIVE_PURIFY_ALARM %
%   N10:4/0  H2_LEAK_ALARM %
%   B36:1/2  PURGE_COMPLETE %
%   N10:2/0  GET_LT_SHUTDOWN_ALM %
%   N10:16/1  SYSTEM_WARNING_FLAG %
%   N10:8/0  SCREEN_COMMS_ERROR %
%   B34:2/1  ACTIVE_REGEN_WARNING %
%   N200:0  HMI_SYSTEM_STATUS %

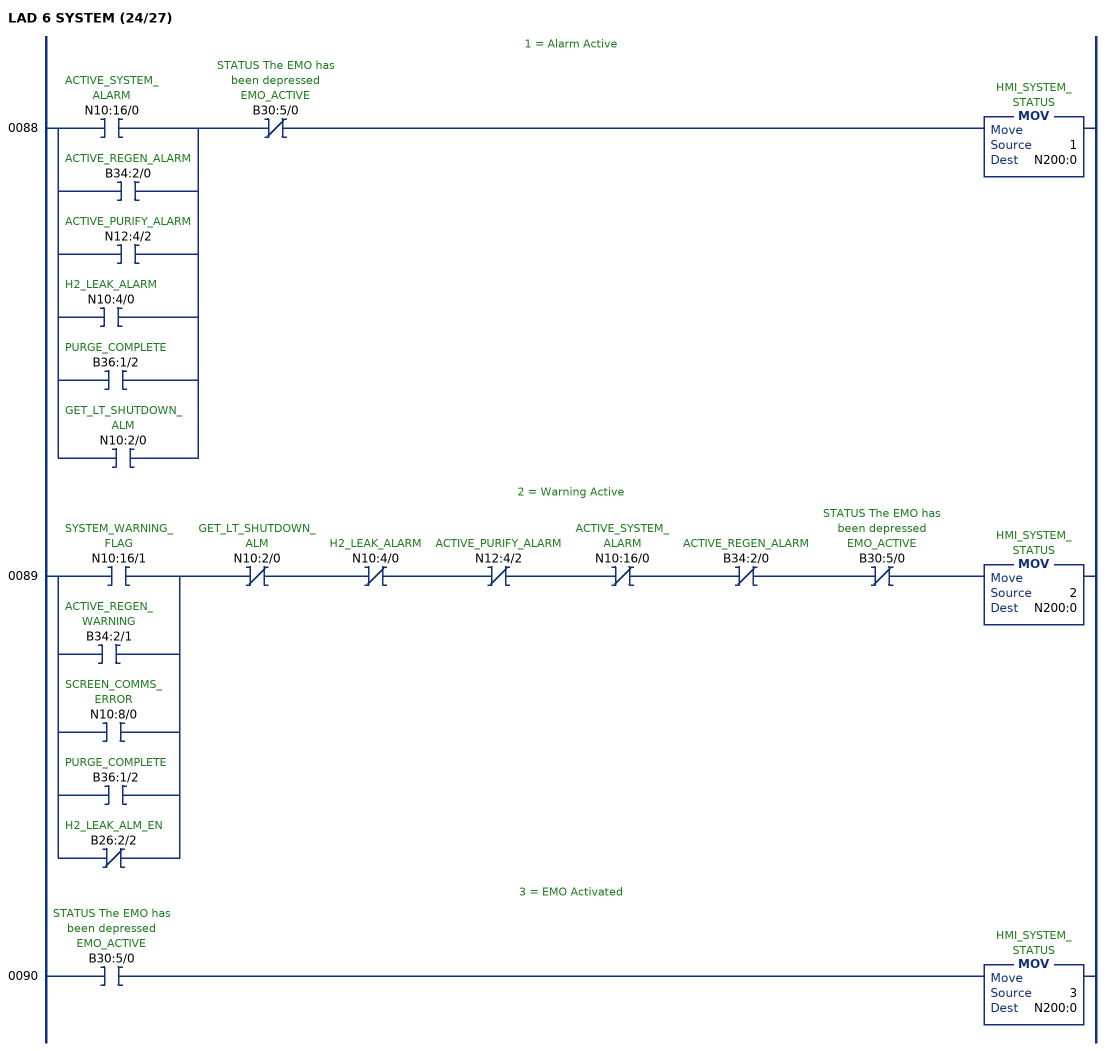
% Rung: 88 %
% 1 = Alarm Active %
SOR BST XIC N10:16/0 NXB XIC B34:2/0 NXB XIC N12:4/2 NXB XIC N10:4/0 NXB XIC B36:1/2 NXB XIC N10:2/0 BND XIO B30:5/0 MOV 1 N200:0 EOR
%   N10:16/0  ACTIVE_SYSTEM_ALARM %
%   B34:2/0  ACTIVE_REGEN_ALARM %
%   N12:4/2  ACTIVE_PURIFY_ALARM %
%   N10:4/0  H2_LEAK_ALARM %
%   B36:1/2  PURGE_COMPLETE %
%   N10:2/0  GET_LT_SHUTDOWN_ALM %
%   B30:5/0  EMO_ACTIVE  "STATUS The EMO has been depressed" %
%   N200:0  HMI_SYSTEM_STATUS %
% Rung: 89 %
% 2 = Warning Active %
SOR BST XIC N10:16/1 NXB XIC B34:2/1 NXB XIC N10:8/0 NXB XIC B36:1/2 NXB XIO B26:2/2 BND XIO N10:2/0 XIO N10:4/0 XIO N12:4/2 XIO N10:16/0 XIO B34:2/0 XIO B30:5/0 MOV 2 N200:0 EOR
%   N10:16/1  SYSTEM_WARNING_FLAG %
%   B34:2/1  ACTIVE_REGEN_WARNING %
%   N10:8/0  SCREEN_COMMS_ERROR %
%   B36:1/2  PURGE_COMPLETE %
%   B26:2/2  H2_LEAK_ALM_EN %
%   N10:2/0  GET_LT_SHUTDOWN_ALM %
%   N10:4/0  H2_LEAK_ALARM %
%   N12:4/2  ACTIVE_PURIFY_ALARM %
%   N10:16/0  ACTIVE_SYSTEM_ALARM %
%   B34:2/0  ACTIVE_REGEN_ALARM %
%   B30:5/0  EMO_ACTIVE  "STATUS The EMO has been depressed" %
%   N200:0  HMI_SYSTEM_STATUS %
% Rung: 90 %
% 3 = EMO Activated %
SOR XIC B30:5/0 MOV 3 N200:0 EOR
%   B30:5/0  EMO_ACTIVE  "STATUS The EMO has been depressed" %
%   N200:0  HMI_SYSTEM_STATUS %

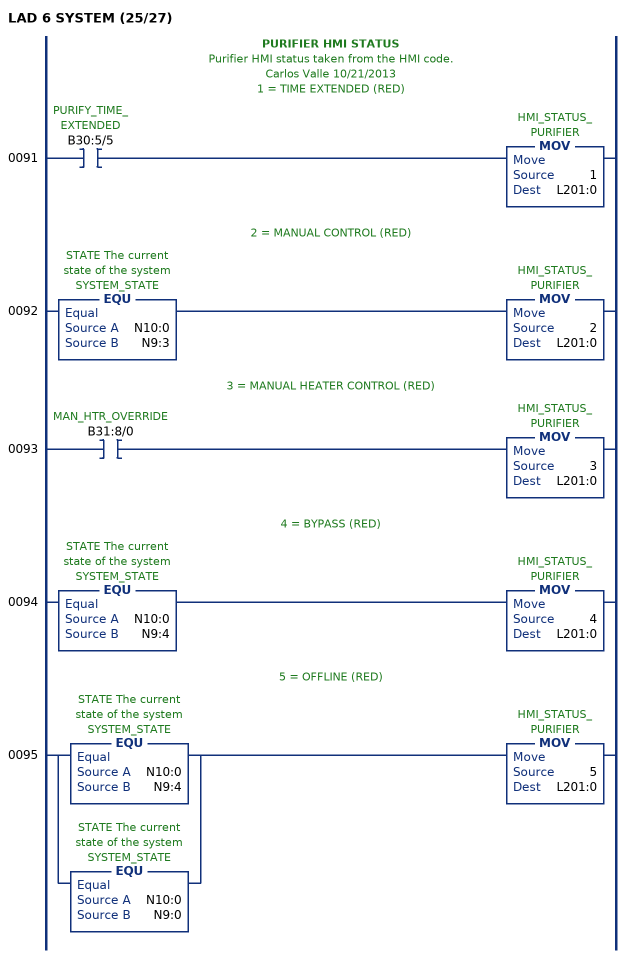
% Rung: 91 %
% TITLE: PURIFIER HMI STATUS %
% Purifier HMI status taken from the HMI code.
% Carlos Valle 10/21/2013
% 1 = TIME EXTENDED (RED) %
SOR XIC B30:5/5 MOV 1 L201:0 EOR
%   B30:5/5  PURIFY_TIME_EXTENDED %
%   L201:0  HMI_STATUS_PURIFIER %
% Rung: 92 %
% 2 = MANUAL CONTROL (RED) %
SOR EQU N10:0 N9:3 MOV 2 L201:0 EOR
%   N10:0  SYSTEM_STATE  "STATE The current state of the system" %
%   N9:3  SYSTEM_MANUAL  "STATE System Manual" %
%   L201:0  HMI_STATUS_PURIFIER %
% Rung: 93 %
% 3 = MANUAL HEATER CONTROL (RED) %
SOR XIC B31:8/0 MOV 3 L201:0 EOR
%   B31:8/0  MAN_HTR_OVERRIDE %
%   L201:0  HMI_STATUS_PURIFIER %
% Rung: 94 %
% 4 = BYPASS (RED) %
SOR EQU N10:0 N9:4 MOV 4 L201:0 EOR
%   N10:0  SYSTEM_STATE  "STATE The current state of the system" %
%   N9:4  SYSTEM_ALARM  "STATE System Alarm" %
%   L201:0  HMI_STATUS_PURIFIER %
% Rung: 95 %
% 5 = OFFLINE (RED) %
SOR BST EQU N10:0 N9:4 NXB EQU N10:0 N9:0 BND MOV 5 L201:0 EOR
%   N10:0  SYSTEM_STATE  "STATE The current state of the system" %
%   N9:4  SYSTEM_ALARM  "STATE System Alarm" %
%   N9:0  SYSTEM_OFFLINE %
%   L201:0  HMI_STATUS_PURIFIER %

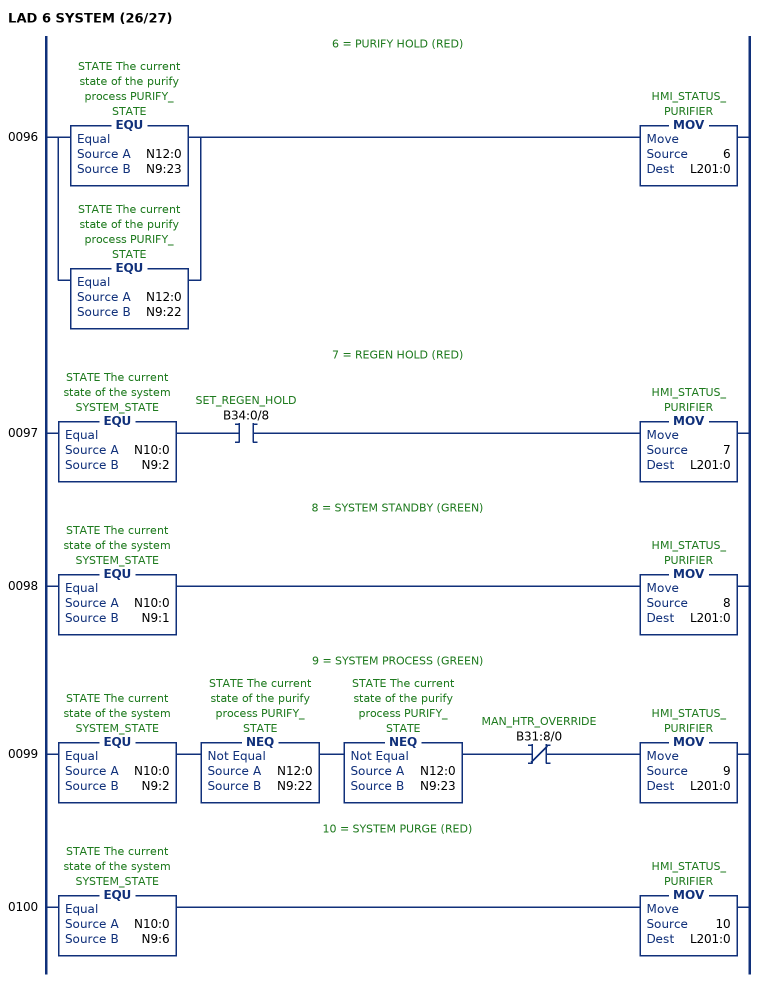
% Rung: 96 %
% 6 = PURIFY HOLD (RED) %
SOR BST EQU N12:0 N9:23 NXB EQU N12:0 N9:22 BND MOV 6 L201:0 EOR
%   N12:0  PURIFY_STATE  "STATE The current state of the purify process" %
%   N9:23  PURIFY_MANUAL_HOLD  "STATE Purify Manual Hold" %
%   N9:22  PURIFY_HOLD  "STATE Purify Hold" %
%   L201:0  HMI_STATUS_PURIFIER %
% Rung: 97 %
% 7 = REGEN HOLD (RED) %
SOR EQU N10:0 N9:2 XIC B34:0/8 MOV 7 L201:0 EOR
%   N10:0  SYSTEM_STATE  "STATE The current state of the system" %
%   N9:2  SYSTEM_PROCESS  "STATE System Process" %
%   B34:0/8  SET_REGEN_HOLD %
%   L201:0  HMI_STATUS_PURIFIER %
% Rung: 98 %
% 8 = SYSTEM STANDBY (GREEN) %
SOR EQU N10:0 N9:1 MOV 8 L201:0 EOR
%   N10:0  SYSTEM_STATE  "STATE The current state of the system" %
%   N9:1  SYSTEM_STANDBY  "STATE System Process" %
%   L201:0  HMI_STATUS_PURIFIER %
% Rung: 99 %
% 9 = SYSTEM PROCESS (GREEN) %
SOR EQU N10:0 N9:2 NEQ N12:0 N9:22 NEQ N12:0 N9:23 XIO B31:8/0 MOV 9 L201:0 EOR
%   N10:0  SYSTEM_STATE  "STATE The current state of the system" %
%   N9:2  SYSTEM_PROCESS  "STATE System Process" %
%   N12:0  PURIFY_STATE  "STATE The current state of the purify process" %
%   N9:22  PURIFY_HOLD  "STATE Purify Hold" %
%   N9:23  PURIFY_MANUAL_HOLD  "STATE Purify Manual Hold" %
%   B31:8/0  MAN_HTR_OVERRIDE %
%   L201:0  HMI_STATUS_PURIFIER %
% Rung: 100 %
% 10 = SYSTEM PURGE (RED) %
SOR EQU N10:0 N9:6 MOV 10 L201:0 EOR
%   N10:0  SYSTEM_STATE  "STATE The current state of the system" %
%   N9:6  SYSTEM_PURGE %
%   L201:0  HMI_STATUS_PURIFIER %

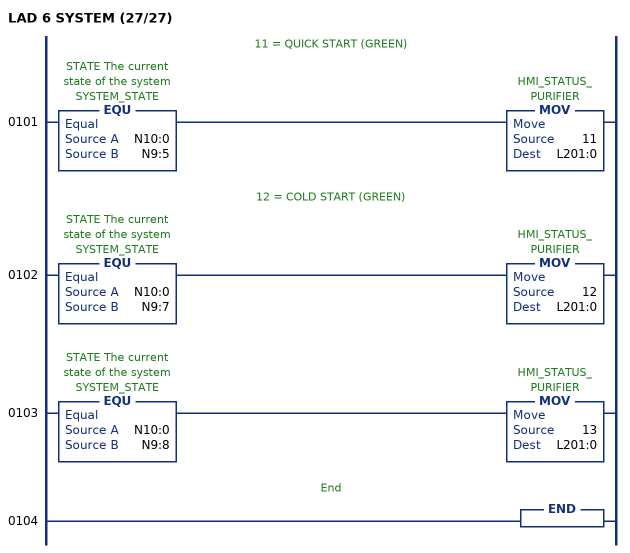
% Rung: 101 %
% 11 = QUICK START (GREEN) %
SOR EQU N10:0 N9:5 MOV 11 L201:0 EOR
%   N10:0  SYSTEM_STATE  "STATE The current state of the system" %
%   N9:5  SYSTEM_QUICK_START %
%   L201:0  HMI_STATUS_PURIFIER %
% Rung: 102 %
% 12 = COLD START (GREEN) %
SOR EQU N10:0 N9:7 MOV 12 L201:0 EOR
%   N10:0  SYSTEM_STATE  "STATE The current state of the system" %
%   N9:7  SYSTEM_COLD_START %
%   L201:0  HMI_STATUS_PURIFIER %
% Rung: 103 %
SOR EQU N10:0 N9:8 MOV 13 L201:0 EOR
%   N10:0  SYSTEM_STATE  "STATE The current state of the system" %
%   N9:8  SYSTEM_SUPPLEMENTAL %
%   L201:0  HMI_STATUS_PURIFIER %
% Rung: 104 %
% End %
SOR END EOR

LADDER 7 "PROCESSING"    % Runs the processing control %
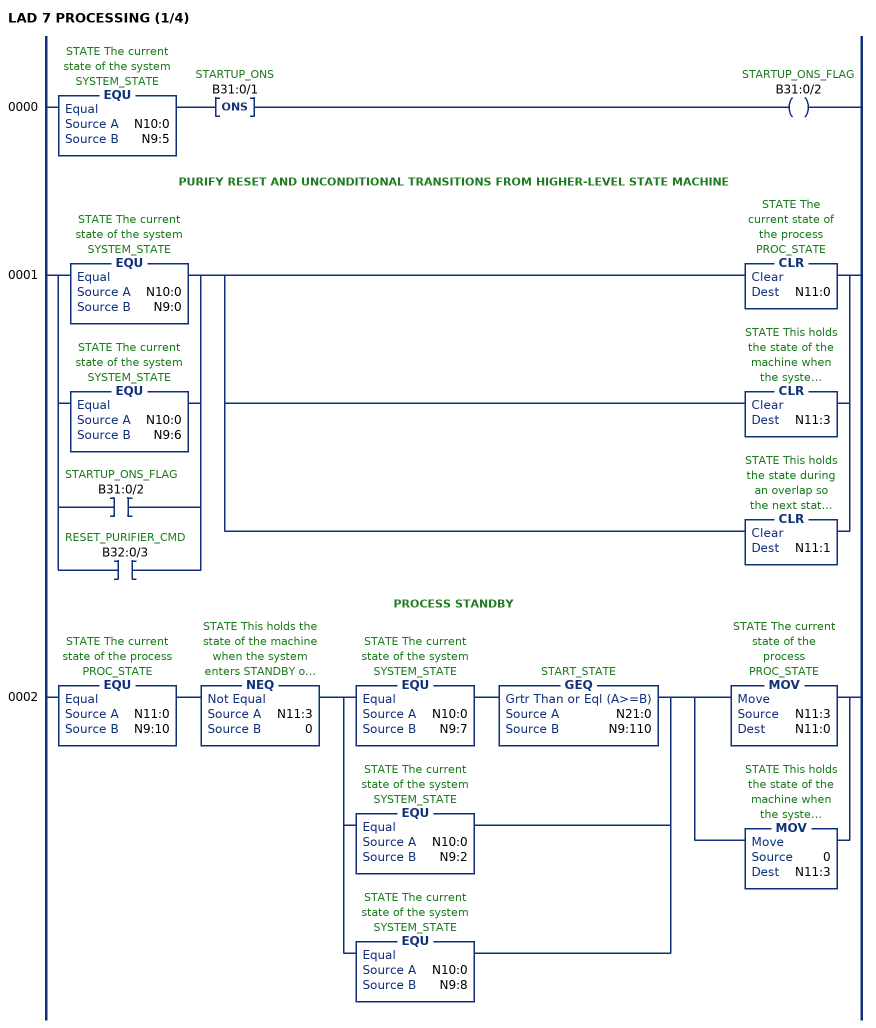
% Rung: 0 %
SOR EQU N10:0 N9:5 ONS B31:0/1 OTE B31:0/2 EOR
%   N10:0  SYSTEM_STATE  "STATE The current state of the system" %
%   N9:5  SYSTEM_QUICK_START %
%   B31:0/1  STARTUP_ONS %
%   B31:0/2  STARTUP_ONS_FLAG %
% Rung: 1 %
% TITLE: PURIFY RESET AND UNCONDITIONAL TRANSITIONS FROM HIGHER-LEVEL STATE MACHINE %
SOR BST EQU N10:0 N9:0 NXB EQU N10:0 N9:6 NXB XIC B31:0/2 NXB XIC B32:0/3 BND BST CLR N11:0 NXB CLR N11:3 NXB CLR N11:1 BND EOR
%   N10:0  SYSTEM_STATE  "STATE The current state of the system" %
%   N9:0  SYSTEM_OFFLINE %
%   N9:6  SYSTEM_PURGE %
%   B31:0/2  STARTUP_ONS_FLAG %
%   B32:0/3  RESET_PURIFIER_CMD %
%   N11:0  PROC_STATE  "STATE The current state of the process" %
%   N11:3  PROC_STATE_BUFFER  "STATE This holds the state of the machine when the system enters STANDBY or ALARM" %
%   N11:1  PROC_OVERLAP_BUFFER  "STATE This holds the state during an overlap so the next state can be determined" %
% Rung: 2 %
% TITLE: PROCESS STANDBY %
SOR EQU N11:0 N9:10 NEQ N11:3 0 BST EQU N10:0 N9:7 GEQ N21:0 N9:110 NXB EQU N10:0 N9:2 NXB EQU N10:0 N9:8 BND BST MOV N11:3 N11:0 NXB MOV 0 N11:3 BND EOR
%   N11:0  PROC_STATE  "STATE The current state of the process" %
%   N9:10  PROC_STANDBY  "STATE Process Standby" %
%   N11:3  PROC_STATE_BUFFER  "STATE This holds the state of the machine when the system enters STANDBY or ALARM" %
%   N10:0  SYSTEM_STATE  "STATE The current state of the system" %
%   N9:7  SYSTEM_COLD_START %
%   N21:0  START_STATE %
%   N9:110  START_REG_VENT %
%   N9:2  SYSTEM_PROCESS  "STATE System Process" %
%   N9:8  SYSTEM_SUPPLEMENTAL %

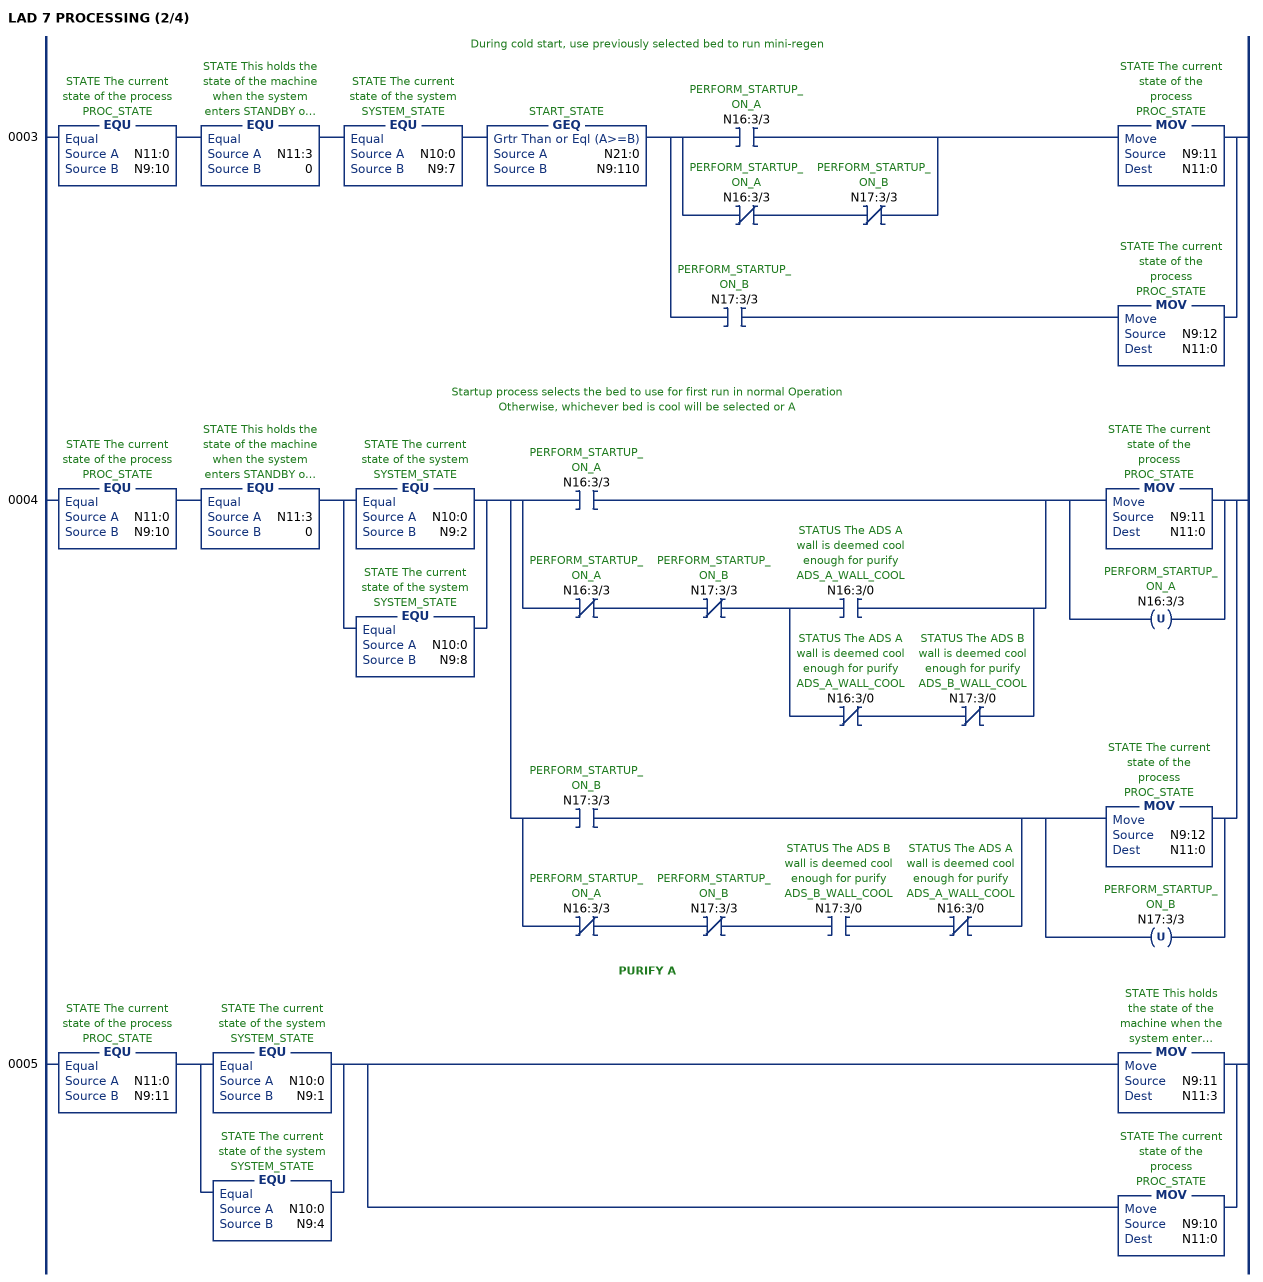
% Rung: 3 %
% During cold start, use previously selected bed to run mini-regen %
SOR EQU N11:0 N9:10 EQU N11:3 0 EQU N10:0 N9:7 GEQ N21:0 N9:110 BST BST XIC N16:3/3 NXB XIO N16:3/3 XIO N17:3/3 BND MOV N9:11 N11:0 NXB XIC N17:3/3 MOV N9:12 N11:0 BND EOR
%   N11:0  PROC_STATE  "STATE The current state of the process" %
%   N9:10  PROC_STANDBY  "STATE Process Standby" %
%   N11:3  PROC_STATE_BUFFER  "STATE This holds the state of the machine when the system enters STANDBY or ALARM" %
%   N10:0  SYSTEM_STATE  "STATE The current state of the system" %
%   N9:7  SYSTEM_COLD_START %
%   N21:0  START_STATE %
%   N9:110  START_REG_VENT %
%   N16:3/3  PERFORM_STARTUP_ON_A %
%   N17:3/3  PERFORM_STARTUP_ON_B %
%   N9:11  PROC_PFY_A_REG_B  "STATE Process Purify A" %
%   N9:12  PROC_PFY_B_REG_A  "STATE Process Purify B" %
% Rung: 4 %
% Startup process selects the bed to use for first run in normal Operation
% Otherwise, whichever bed is cool will be selected or A %
SOR EQU N11:0 N9:10 EQU N11:3 0 BST EQU N10:0 N9:2 NXB EQU N10:0 N9:8 BND BST BST XIC N16:3/3 NXB XIO N16:3/3 XIO N17:3/3 BST XIC N16:3/0 NXB XIO N16:3/0 XIO N17:3/0 BND BND BST MOV N9:11 N11:0 NXB OTU N16:3/3 BND NXB BST XIC N17:3/3 NXB XIO N16:3/3 XIO N17:3/3 XIC N17:3/0 XIO N16:3/0 BND BST MOV N9:12 N11:0 NXB OTU N17:3/3 BND BND EOR
%   N11:0  PROC_STATE  "STATE The current state of the process" %
%   N9:10  PROC_STANDBY  "STATE Process Standby" %
%   N11:3  PROC_STATE_BUFFER  "STATE This holds the state of the machine when the system enters STANDBY or ALARM" %
%   N10:0  SYSTEM_STATE  "STATE The current state of the system" %
%   N9:2  SYSTEM_PROCESS  "STATE System Process" %
%   N9:8  SYSTEM_SUPPLEMENTAL %
%   N16:3/3  PERFORM_STARTUP_ON_A %
%   N17:3/3  PERFORM_STARTUP_ON_B %
%   N16:3/0  ADS_A_WALL_COOL  "STATUS The ADS A wall is deemed cool enough for purify" %
%   N17:3/0  ADS_B_WALL_COOL  "STATUS The ADS B wall is deemed cool enough for purify" %
%   N9:11  PROC_PFY_A_REG_B  "STATE Process Purify A" %
%   N9:12  PROC_PFY_B_REG_A  "STATE Process Purify B" %
% Rung: 5 %
% TITLE: PURIFY A %
SOR EQU N11:0 N9:11 BST EQU N10:0 N9:1 NXB EQU N10:0 N9:4 BND BST MOV N9:11 N11:3 NXB MOV N9:10 N11:0 BND EOR
%   N11:0  PROC_STATE  "STATE The current state of the process" %
%   N9:11  PROC_PFY_A_REG_B  "STATE Process Purify A" %
%   N10:0  SYSTEM_STATE  "STATE The current state of the system" %
%   N9:1  SYSTEM_STANDBY  "STATE System Process" %
%   N9:4  SYSTEM_ALARM  "STATE System Alarm" %
%   N11:3  PROC_STATE_BUFFER  "STATE This holds the state of the machine when the system enters STANDBY or ALARM" %
%   N9:10  PROC_STANDBY  "STATE Process Standby" %

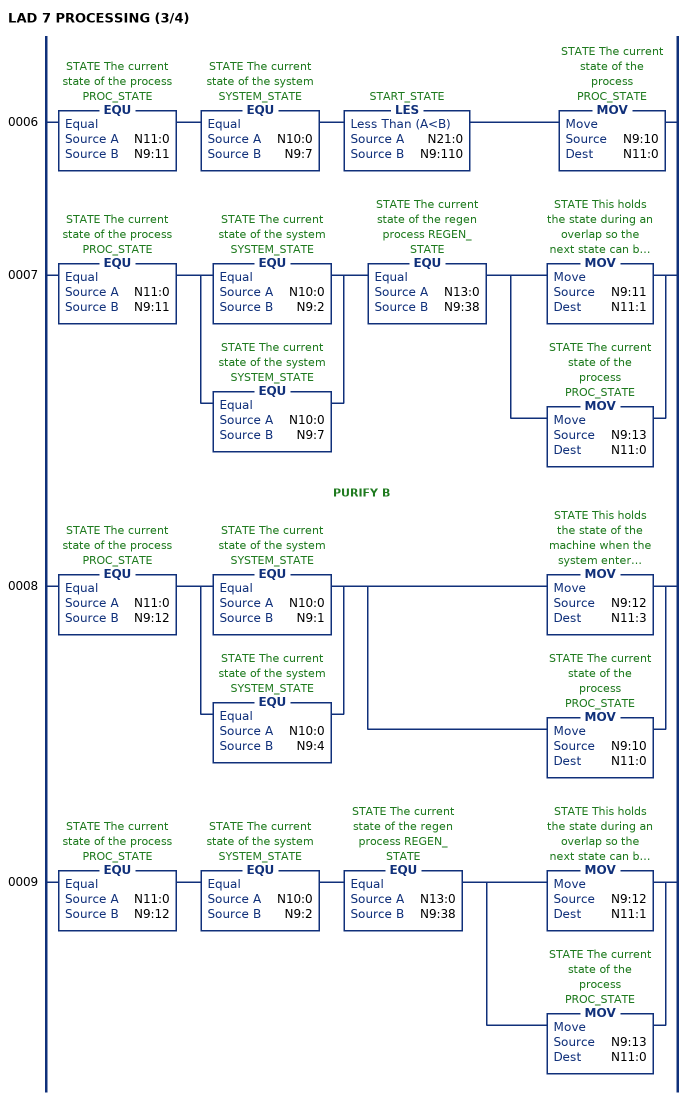
% Rung: 6 %
SOR EQU N11:0 N9:11 EQU N10:0 N9:7 LES N21:0 N9:110 MOV N9:10 N11:0 EOR
%   N11:0  PROC_STATE  "STATE The current state of the process" %
%   N9:11  PROC_PFY_A_REG_B  "STATE Process Purify A" %
%   N10:0  SYSTEM_STATE  "STATE The current state of the system" %
%   N9:7  SYSTEM_COLD_START %
%   N21:0  START_STATE %
%   N9:110  START_REG_VENT %
%   N9:10  PROC_STANDBY  "STATE Process Standby" %
% Rung: 7 %
SOR EQU N11:0 N9:11 BST EQU N10:0 N9:2 NXB EQU N10:0 N9:7 BND EQU N13:0 N9:38 BST MOV N9:11 N11:1 NXB MOV N9:13 N11:0 BND EOR
%   N11:0  PROC_STATE  "STATE The current state of the process" %
%   N9:11  PROC_PFY_A_REG_B  "STATE Process Purify A" %
%   N10:0  SYSTEM_STATE  "STATE The current state of the system" %
%   N9:2  SYSTEM_PROCESS  "STATE System Process" %
%   N9:7  SYSTEM_COLD_START %
%   N13:0  REGEN_STATE  "STATE The current state of the regen process" %
%   N9:38  REGEN_DONE %
%   N11:1  PROC_OVERLAP_BUFFER  "STATE This holds the state during an overlap so the next state can be determined" %
%   N9:13  PROC_OVERLAP  "STATE Process Purify Overlap" %
% Rung: 8 %
% TITLE: PURIFY B %
SOR EQU N11:0 N9:12 BST EQU N10:0 N9:1 NXB EQU N10:0 N9:4 BND BST MOV N9:12 N11:3 NXB MOV N9:10 N11:0 BND EOR
%   N11:0  PROC_STATE  "STATE The current state of the process" %
%   N9:12  PROC_PFY_B_REG_A  "STATE Process Purify B" %
%   N10:0  SYSTEM_STATE  "STATE The current state of the system" %
%   N9:1  SYSTEM_STANDBY  "STATE System Process" %
%   N9:4  SYSTEM_ALARM  "STATE System Alarm" %
%   N11:3  PROC_STATE_BUFFER  "STATE This holds the state of the machine when the system enters STANDBY or ALARM" %
%   N9:10  PROC_STANDBY  "STATE Process Standby" %
% Rung: 9 %
SOR EQU N11:0 N9:12 EQU N10:0 N9:2 EQU N13:0 N9:38 BST MOV N9:12 N11:1 NXB MOV N9:13 N11:0 BND EOR
%   N11:0  PROC_STATE  "STATE The current state of the process" %
%   N9:12  PROC_PFY_B_REG_A  "STATE Process Purify B" %
%   N10:0  SYSTEM_STATE  "STATE The current state of the system" %
%   N9:2  SYSTEM_PROCESS  "STATE System Process" %
%   N13:0  REGEN_STATE  "STATE The current state of the regen process" %
%   N9:38  REGEN_DONE %
%   N11:1  PROC_OVERLAP_BUFFER  "STATE This holds the state during an overlap so the next state can be determined" %
%   N9:13  PROC_OVERLAP  "STATE Process Purify Overlap" %

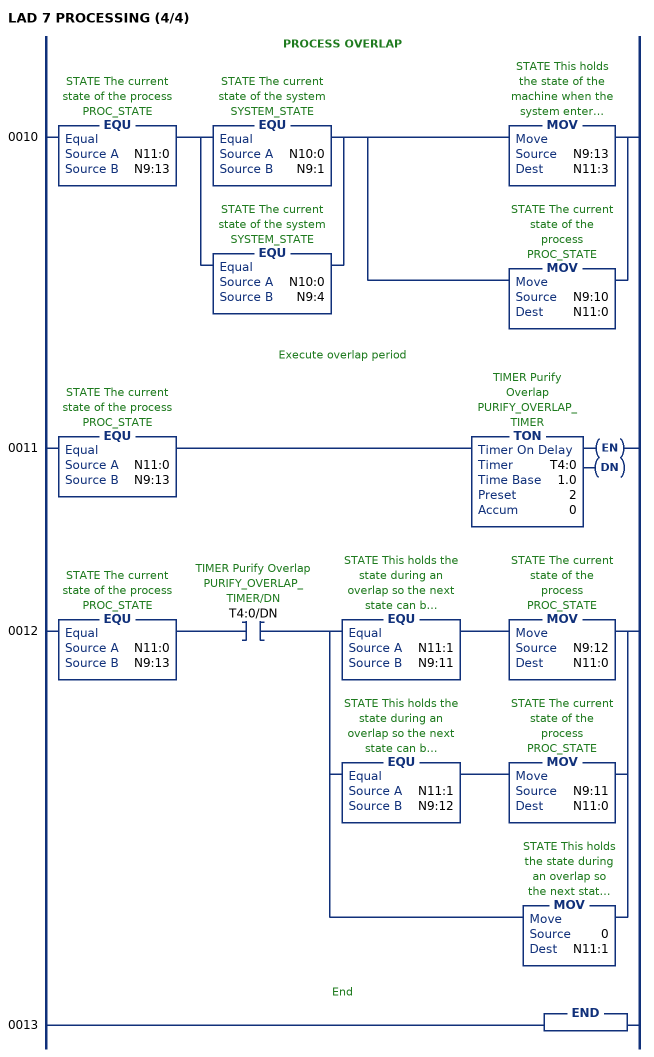
% Rung: 10 %
% TITLE: PROCESS OVERLAP %
SOR EQU N11:0 N9:13 BST EQU N10:0 N9:1 NXB EQU N10:0 N9:4 BND BST MOV N9:13 N11:3 NXB MOV N9:10 N11:0 BND EOR
%   N11:0  PROC_STATE  "STATE The current state of the process" %
%   N9:13  PROC_OVERLAP  "STATE Process Purify Overlap" %
%   N10:0  SYSTEM_STATE  "STATE The current state of the system" %
%   N9:1  SYSTEM_STANDBY  "STATE System Process" %
%   N9:4  SYSTEM_ALARM  "STATE System Alarm" %
%   N11:3  PROC_STATE_BUFFER  "STATE This holds the state of the machine when the system enters STANDBY or ALARM" %
%   N9:10  PROC_STANDBY  "STATE Process Standby" %
% Rung: 11 %
% Execute overlap period %
SOR EQU N11:0 N9:13 TON T4:0 1.0 2 0 EOR
%   N11:0  PROC_STATE  "STATE The current state of the process" %
%   N9:13  PROC_OVERLAP  "STATE Process Purify Overlap" %
%   T4:0  PURIFY_OVERLAP_TIMER  "TIMER Purify Overlap" %
% Rung: 12 %
SOR EQU N11:0 N9:13 XIC T4:0/DN BST EQU N11:1 N9:11 MOV N9:12 N11:0 NXB EQU N11:1 N9:12 MOV N9:11 N11:0 NXB MOV 0 N11:1 BND EOR
%   N11:0  PROC_STATE  "STATE The current state of the process" %
%   N9:13  PROC_OVERLAP  "STATE Process Purify Overlap" %
%   T4:0  PURIFY_OVERLAP_TIMER  "TIMER Purify Overlap" %
%   N11:1  PROC_OVERLAP_BUFFER  "STATE This holds the state during an overlap so the next state can be determined" %
%   N9:11  PROC_PFY_A_REG_B  "STATE Process Purify A" %
%   N9:12  PROC_PFY_B_REG_A  "STATE Process Purify B" %
% Rung: 13 %
% End %
SOR END EOR

LADDER 8 "MANUAL_CTL"    % Runs the manual valve control %
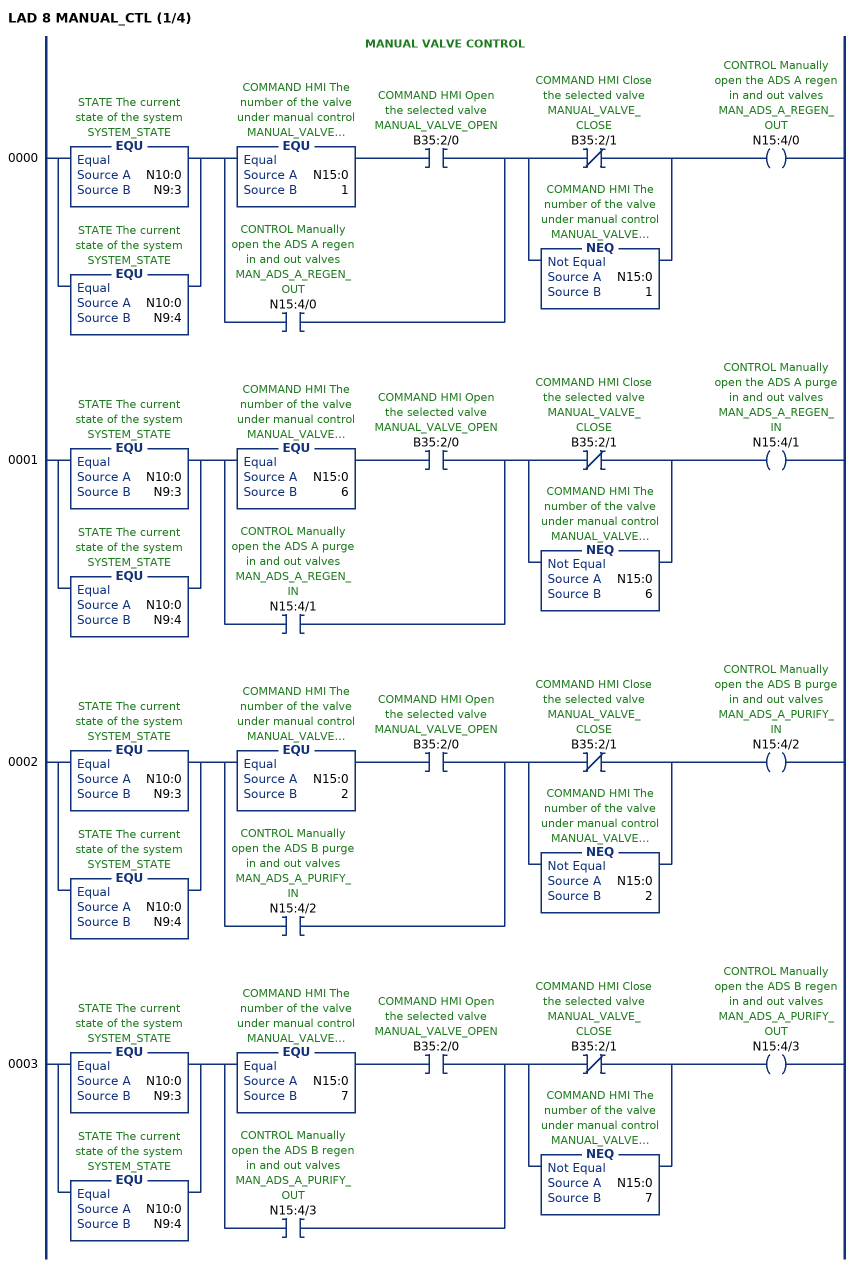
% Rung: 0 %
% TITLE: MANUAL VALVE CONTROL %
SOR BST EQU N10:0 N9:3 NXB EQU N10:0 N9:4 BND BST EQU N15:0 1 XIC B35:2/0 NXB XIC N15:4/0 BND BST XIO B35:2/1 NXB NEQ N15:0 1 BND OTE N15:4/0 EOR
%   N10:0  SYSTEM_STATE  "STATE The current state of the system" %
%   N9:3  SYSTEM_MANUAL  "STATE System Manual" %
%   N9:4  SYSTEM_ALARM  "STATE System Alarm" %
%   N15:0  MANUAL_VALVE_NUMBER  "COMMAND HMI The number of the valve under manual control" %
%   B35:2/0  MANUAL_VALVE_OPEN  "COMMAND HMI Open the selected valve" %
%   N15:4/0  MAN_ADS_A_REGEN_OUT  "CONTROL Manually open the ADS A regen in and out valves" %
%   B35:2/1  MANUAL_VALVE_CLOSE  "COMMAND HMI Close the selected valve" %
% Rung: 1 %
SOR BST EQU N10:0 N9:3 NXB EQU N10:0 N9:4 BND BST EQU N15:0 6 XIC B35:2/0 NXB XIC N15:4/1 BND BST XIO B35:2/1 NXB NEQ N15:0 6 BND OTE N15:4/1 EOR
%   N10:0  SYSTEM_STATE  "STATE The current state of the system" %
%   N9:3  SYSTEM_MANUAL  "STATE System Manual" %
%   N9:4  SYSTEM_ALARM  "STATE System Alarm" %
%   N15:0  MANUAL_VALVE_NUMBER  "COMMAND HMI The number of the valve under manual control" %
%   B35:2/0  MANUAL_VALVE_OPEN  "COMMAND HMI Open the selected valve" %
%   N15:4/1  MAN_ADS_A_REGEN_IN  "CONTROL Manually open the ADS A purge in and out valves" %
%   B35:2/1  MANUAL_VALVE_CLOSE  "COMMAND HMI Close the selected valve" %
% Rung: 2 %
SOR BST EQU N10:0 N9:3 NXB EQU N10:0 N9:4 BND BST EQU N15:0 2 XIC B35:2/0 NXB XIC N15:4/2 BND BST XIO B35:2/1 NXB NEQ N15:0 2 BND OTE N15:4/2 EOR
%   N10:0  SYSTEM_STATE  "STATE The current state of the system" %
%   N9:3  SYSTEM_MANUAL  "STATE System Manual" %
%   N9:4  SYSTEM_ALARM  "STATE System Alarm" %
%   N15:0  MANUAL_VALVE_NUMBER  "COMMAND HMI The number of the valve under manual control" %
%   B35:2/0  MANUAL_VALVE_OPEN  "COMMAND HMI Open the selected valve" %
%   N15:4/2  MAN_ADS_A_PURIFY_IN  "CONTROL Manually open the ADS B purge in and out valves" %
%   B35:2/1  MANUAL_VALVE_CLOSE  "COMMAND HMI Close the selected valve" %
% Rung: 3 %
SOR BST EQU N10:0 N9:3 NXB EQU N10:0 N9:4 BND BST EQU N15:0 7 XIC B35:2/0 NXB XIC N15:4/3 BND BST XIO B35:2/1 NXB NEQ N15:0 7 BND OTE N15:4/3 EOR
%   N10:0  SYSTEM_STATE  "STATE The current state of the system" %
%   N9:3  SYSTEM_MANUAL  "STATE System Manual" %
%   N9:4  SYSTEM_ALARM  "STATE System Alarm" %
%   N15:0  MANUAL_VALVE_NUMBER  "COMMAND HMI The number of the valve under manual control" %
%   B35:2/0  MANUAL_VALVE_OPEN  "COMMAND HMI Open the selected valve" %
%   N15:4/3  MAN_ADS_A_PURIFY_OUT  "CONTROL Manually open the ADS B regen in and out valves" %
%   B35:2/1  MANUAL_VALVE_CLOSE  "COMMAND HMI Close the selected valve" %

